   AI_RAW_8701.___________0040_1 := false;
   AI_RAW_8701.___________0040_2 := false;
   AI_RAW_8701.VALUE_COEF := 0.00617;
   AI_RAW_8801.revInfo.REV_BLOCK := 'UT00801';
   AI_RAW_8801.revInfo.REV_NUMBER := '001.000';
   AI_RAW_8801.revInfo.REV_DATE := '2024-04-09';
   AI_RAW_8801.revInfo.REV_AUTHOR := 'M. Gledhill';
   AI_RAW_8801.___________0010_0 := false;
   AI_RAW_8801.___________0010_1 := false;
   AI_RAW_8801.AI_CODE := 16#8801;
   AI_RAW_8801.___________0020_0 := false;
   AI_RAW_8801.___________0020_1 := false;
   AI_RAW_8801.RAW_MIN := -6000;
   AI_RAW_8801.RAW_MAX := 13000;
   AI_RAW_8801.RAW_DESC := 'Thermal Resistance - 3-wire (Ni100 climate - 618)';
   AI_RAW_8801.___________0030_1 := false;
   AI_RAW_8801.___________0030_2 := false;
   AI_RAW_8801.PARAM_TYPE := 16#08;
   AI_RAW_8801.PARAM_RANGE := 16#01;
   AI_RAW_8801.PARAM_COEF := 16#08;
   AI_RAW_8801.___________0040_1 := false;
   AI_RAW_8801.___________0040_2 := false;
   AI_RAW_8801.VALUE_COEF := 0.00618;
   AI_RAW_8901.revInfo.REV_BLOCK := 'UT00801';
   AI_RAW_8901.revInfo.REV_NUMBER := '001.000';
   AI_RAW_8901.revInfo.REV_DATE := '2024-04-09';
   AI_RAW_8901.revInfo.REV_AUTHOR := 'M. Gledhill';
   AI_RAW_8901.___________0010_0 := false;
   AI_RAW_8901.___________0010_1 := false;
   AI_RAW_8901.AI_CODE := 16#8901;
   AI_RAW_8901.___________0020_0 := false;
   AI_RAW_8901.___________0020_1 := false;
   AI_RAW_8901.RAW_MIN := -6000;
   AI_RAW_8901.RAW_MAX := 13000;
   AI_RAW_8901.RAW_DESC := 'Thermal Resistance - 3-wire (Ni100 climate - 672)';
   AI_RAW_8901.___________0030_1 := false;
   AI_RAW_8901.___________0030_2 := false;
   AI_RAW_8901.PARAM_TYPE := 16#08;
   AI_RAW_8901.PARAM_RANGE := 16#01;
   AI_RAW_8901.PARAM_COEF := 16#09;
   AI_RAW_8901.___________0040_1 := false;
   AI_RAW_8901.___________0040_2 := false;
   AI_RAW_8901.VALUE_COEF := 0.00672;
   AI_RAW_8703.revInfo.REV_BLOCK := 'UT00801';
   AI_RAW_8703.revInfo.REV_NUMBER := '001.000';
   AI_RAW_8703.revInfo.REV_DATE := '2024-04-09';
   AI_RAW_8703.revInfo.REV_AUTHOR := 'M. Gledhill';
   AI_RAW_8703.___________0010_0 := false;
   AI_RAW_8703.___________0010_1 := false;
   AI_RAW_8703.AI_CODE := 16#8703;
   AI_RAW_8703.___________0020_0 := false;
   AI_RAW_8703.___________0020_1 := false;
   AI_RAW_8703.RAW_MIN := -600;
   AI_RAW_8703.RAW_MAX := 1800;
   AI_RAW_8703.RAW_DESC := 'Thermal Resistance - 3-wire (Ni100 standard - 617)';
   AI_RAW_8703.___________0030_1 := false;
   AI_RAW_8703.___________0030_2 := false;
   AI_RAW_8703.PARAM_TYPE := 16#08;
   AI_RAW_8703.PARAM_RANGE := 16#03;
   AI_RAW_8703.PARAM_COEF := 16#07;
   AI_RAW_8703.___________0040_1 := false;
   AI_RAW_8703.___________0040_2 := false;
   AI_RAW_8703.VALUE_COEF := 0.00617;
   AI_RAW_8803.revInfo.REV_BLOCK := 'UT00801';
   AI_RAW_8803.revInfo.REV_NUMBER := '001.000';
   AI_RAW_8803.revInfo.REV_DATE := '2024-04-09';
   AI_RAW_8803.revInfo.REV_AUTHOR := 'M. Gledhill';
   AI_RAW_8803.___________0010_0 := false;
   AI_RAW_8803.___________0010_1 := false;
   AI_RAW_8803.AI_CODE := 16#8803;
   AI_RAW_8803.___________0020_0 := false;
   AI_RAW_8803.___________0020_1 := false;
   AI_RAW_8803.RAW_MIN := -600;
   AI_RAW_8803.RAW_MAX := 2500;
   AI_RAW_8803.RAW_DESC := 'Thermal Resistance - 3-wire (Ni100 standard - 618)';
   AI_RAW_8803.___________0030_1 := false;
   AI_RAW_8803.___________0030_2 := false;
   AI_RAW_8803.PARAM_TYPE := 16#08;
   AI_RAW_8803.PARAM_RANGE := 16#03;
   AI_RAW_8803.PARAM_COEF := 16#08;
   AI_RAW_8803.___________0040_1 := false;
   AI_RAW_8803.___________0040_2 := false;
   AI_RAW_8803.VALUE_COEF := 0.00618;
   AI_RAW_8903.revInfo.REV_BLOCK := 'UT00801';
   AI_RAW_8903.revInfo.REV_NUMBER := '001.000';
   AI_RAW_8903.revInfo.REV_DATE := '2024-04-09';
   AI_RAW_8903.revInfo.REV_AUTHOR := 'M. Gledhill';
   AI_RAW_8903.___________0010_0 := false;
   AI_RAW_8903.___________0010_1 := false;
   AI_RAW_8903.AI_CODE := 16#8903;
   AI_RAW_8903.___________0020_0 := false;
   AI_RAW_8903.___________0020_1 := false;
   AI_RAW_8903.RAW_MIN := -600;
   AI_RAW_8903.RAW_MAX := 2500;
   AI_RAW_8903.RAW_DESC := 'Thermal Resistance - 3-wire (Ni100 standard - 672)';
   AI_RAW_8903.___________0030_1 := false;
   AI_RAW_8903.___________0030_2 := false;
   AI_RAW_8903.PARAM_TYPE := 16#08;
   AI_RAW_8903.PARAM_RANGE := 16#03;
   AI_RAW_8903.PARAM_COEF := 16#09;
   AI_RAW_8903.___________0040_1 := false;
   AI_RAW_8903.___________0040_2 := false;
   AI_RAW_8903.VALUE_COEF := 0.00672;
   AI_RAW_8711.revInfo.REV_BLOCK := 'UT00801';
   AI_RAW_8711.revInfo.REV_NUMBER := '001.000';
   AI_RAW_8711.revInfo.REV_DATE := '2024-04-09';
   AI_RAW_8711.revInfo.REV_AUTHOR := 'M. Gledhill';
   AI_RAW_8711.___________0010_0 := false;
   AI_RAW_8711.___________0010_1 := false;
   AI_RAW_8711.AI_CODE := 16#8711;
   AI_RAW_8711.___________0020_0 := false;
   AI_RAW_8711.___________0020_1 := false;
   AI_RAW_8711.RAW_MIN := -6000;
   AI_RAW_8711.RAW_MAX := 13000;
   AI_RAW_8711.RAW_DESC := 'Thermal Resistance - 3-wire (Ni200 climate - 617)';
   AI_RAW_8711.___________0030_1 := false;
   AI_RAW_8711.___________0030_2 := false;
   AI_RAW_8711.PARAM_TYPE := 16#08;
   AI_RAW_8711.PARAM_RANGE := 16#11;
   AI_RAW_8711.PARAM_COEF := 16#07;
   AI_RAW_8711.___________0040_1 := false;
   AI_RAW_8711.___________0040_2 := false;
   AI_RAW_8711.VALUE_COEF := 0.00617;
   AI_RAW_8811.revInfo.REV_BLOCK := 'UT00801';
   AI_RAW_8811.revInfo.REV_NUMBER := '001.000';
   AI_RAW_8811.revInfo.REV_DATE := '2024-04-09';
   AI_RAW_8811.revInfo.REV_AUTHOR := 'M. Gledhill';
   AI_RAW_8811.___________0010_0 := false;
   AI_RAW_8811.___________0010_1 := false;
   AI_RAW_8811.AI_CODE := 16#8811;
   AI_RAW_8811.___________0020_0 := false;
   AI_RAW_8811.___________0020_1 := false;
   AI_RAW_8811.RAW_MIN := -6000;
   AI_RAW_8811.RAW_MAX := 13000;
   AI_RAW_8811.RAW_DESC := 'Thermal Resistance - 3-wire (Ni200 climate - 618)';
   AI_RAW_8811.___________0030_1 := false;
   AI_RAW_8811.___________0030_2 := false;
   AI_RAW_8811.PARAM_TYPE := 16#08;
   AI_RAW_8811.PARAM_RANGE := 16#11;
   AI_RAW_8811.PARAM_COEF := 16#08;
   AI_RAW_8811.___________0040_1 := false;
   AI_RAW_8811.___________0040_2 := false;
   AI_RAW_8811.VALUE_COEF := 0.00618;
   AI_RAW_8911.revInfo.REV_BLOCK := 'UT00801';
   AI_RAW_8911.revInfo.REV_NUMBER := '001.000';
   AI_RAW_8911.revInfo.REV_DATE := '2024-04-09';
   AI_RAW_8911.revInfo.REV_AUTHOR := 'M. Gledhill';
   AI_RAW_8911.___________0010_0 := false;
   AI_RAW_8911.___________0010_1 := false;
   AI_RAW_8911.AI_CODE := 16#8911;
   AI_RAW_8911.___________0020_0 := false;
   AI_RAW_8911.___________0020_1 := false;
   AI_RAW_8911.RAW_MIN := -6000;
   AI_RAW_8911.RAW_MAX := 13000;
   AI_RAW_8911.RAW_DESC := 'Thermal Resistance - 3-wire (Ni200 climate - 672)';
   AI_RAW_8911.___________0030_1 := false;
   AI_RAW_8911.___________0030_2 := false;
   AI_RAW_8911.PARAM_TYPE := 16#08;
   AI_RAW_8911.PARAM_RANGE := 16#11;
   AI_RAW_8911.PARAM_COEF := 16#09;
   AI_RAW_8911.___________0040_1 := false;
   AI_RAW_8911.___________0040_2 := false;
   AI_RAW_8911.VALUE_COEF := 0.00672;
   AI_RAW_8710.revInfo.REV_BLOCK := 'UT00801';
   AI_RAW_8710.revInfo.REV_NUMBER := '001.000';
   AI_RAW_8710.revInfo.REV_DATE := '2024-04-09';
   AI_RAW_8710.revInfo.REV_AUTHOR := 'M. Gledhill';
   AI_RAW_8710.___________0010_0 := false;
   AI_RAW_8710.___________0010_1 := false;
   AI_RAW_8710.AI_CODE := 16#8710;
   AI_RAW_8710.___________0020_0 := false;
   AI_RAW_8710.___________0020_1 := false;
   AI_RAW_8710.RAW_MIN := -600;
   AI_RAW_8710.RAW_MAX := 1800;
   AI_RAW_8710.RAW_DESC := 'Thermal Resistance - 3-wire (Ni200 standard - 617)';
   AI_RAW_8710.___________0030_1 := false;
   AI_RAW_8710.___________0030_2 := false;
   AI_RAW_8710.PARAM_TYPE := 16#08;
   AI_RAW_8710.PARAM_RANGE := 16#10;
   AI_RAW_8710.PARAM_COEF := 16#07;
   AI_RAW_8710.___________0040_1 := false;
   AI_RAW_8710.___________0040_2 := false;
   AI_RAW_8710.VALUE_COEF := 0.00617;
   AI_RAW_8810.revInfo.REV_BLOCK := 'UT00801';
   AI_RAW_8810.revInfo.REV_NUMBER := '001.000';
   AI_RAW_8810.revInfo.REV_DATE := '2024-04-09';
   AI_RAW_8810.revInfo.REV_AUTHOR := 'M. Gledhill';
   AI_RAW_8810.___________0010_0 := false;
   AI_RAW_8810.___________0010_1 := false;
   AI_RAW_8810.AI_CODE := 16#8810;
   AI_RAW_8810.___________0020_0 := false;
   AI_RAW_8810.___________0020_1 := false;
   AI_RAW_8810.RAW_MIN := -600;
   AI_RAW_8810.RAW_MAX := 2500;
   AI_RAW_8810.RAW_DESC := 'Thermal Resistance - 3-wire (Ni200 standard - 618)';
   AI_RAW_8810.___________0030_1 := false;
   AI_RAW_8810.___________0030_2 := false;
   AI_RAW_8810.PARAM_TYPE := 16#08;
   AI_RAW_8810.PARAM_RANGE := 16#10;
   AI_RAW_8810.PARAM_COEF := 16#08;
   AI_RAW_8810.___________0040_1 := false;
   AI_RAW_8810.___________0040_2 := false;
   AI_RAW_8810.VALUE_COEF := 0.00618;
   AI_RAW_8910.revInfo.REV_BLOCK := 'UT00801';
   AI_RAW_8910.revInfo.REV_NUMBER := '001.000';
   AI_RAW_8910.revInfo.REV_DATE := '2024-04-09';
   AI_RAW_8910.revInfo.REV_AUTHOR := 'M. Gledhill';
   AI_RAW_8910.___________0010_0 := false;
   AI_RAW_8910.___________0010_1 := false;
   AI_RAW_8910.AI_CODE := 16#8910;
   AI_RAW_8910.___________0020_0 := false;
   AI_RAW_8910.___________0020_1 := false;
   AI_RAW_8910.RAW_MIN := -600;
   AI_RAW_8910.RAW_MAX := 2500;
   AI_RAW_8910.RAW_DESC := 'Thermal Resistance - 3-wire (Ni200 standard - 672)';
   AI_RAW_8910.___________0030_1 := false;
   AI_RAW_8910.___________0030_2 := false;
   AI_RAW_8910.PARAM_TYPE := 16#08;
   AI_RAW_8910.PARAM_RANGE := 16#10;
   AI_RAW_8910.PARAM_COEF := 16#09;
   AI_RAW_8910.___________0040_1 := false;
   AI_RAW_8910.___________0040_2 := false;
   AI_RAW_8910.VALUE_COEF := 0.00672;
   AI_RAW_8713.revInfo.REV_BLOCK := 'UT00801';
   AI_RAW_8713.revInfo.REV_NUMBER := '001.000';
   AI_RAW_8713.revInfo.REV_DATE := '2024-04-09';
   AI_RAW_8713.revInfo.REV_AUTHOR := 'M. Gledhill';
   AI_RAW_8713.___________0010_0 := false;
   AI_RAW_8713.___________0010_1 := false;
   AI_RAW_8713.AI_CODE := 16#8713;
   AI_RAW_8713.___________0020_0 := false;
   AI_RAW_8713.___________0020_1 := false;
   AI_RAW_8713.RAW_MIN := -6000;
   AI_RAW_8713.RAW_MAX := 13000;
   AI_RAW_8713.RAW_DESC := 'Thermal Resistance - 3-wire (Ni500 climate - 617)';
   AI_RAW_8713.___________0030_1 := false;
   AI_RAW_8713.___________0030_2 := false;
   AI_RAW_8713.PARAM_TYPE := 16#08;
   AI_RAW_8713.PARAM_RANGE := 16#13;
   AI_RAW_8713.PARAM_COEF := 16#07;
   AI_RAW_8713.___________0040_1 := false;
   AI_RAW_8713.___________0040_2 := false;
   AI_RAW_8713.VALUE_COEF := 0.00617;
   AI_RAW_8813.revInfo.REV_BLOCK := 'UT00801';
   AI_RAW_8813.revInfo.REV_NUMBER := '001.000';
   AI_RAW_8813.revInfo.REV_DATE := '2024-04-09';
   AI_RAW_8813.revInfo.REV_AUTHOR := 'M. Gledhill';
   AI_RAW_8813.___________0010_0 := false;
   AI_RAW_8813.___________0010_1 := false;
   AI_RAW_8813.AI_CODE := 16#8813;
   AI_RAW_8813.___________0020_0 := false;
   AI_RAW_8813.___________0020_1 := false;
   AI_RAW_8813.RAW_MIN := -6000;
   AI_RAW_8813.RAW_MAX := 13000;
   AI_RAW_8813.RAW_DESC := 'Thermal Resistance - 3-wire (Ni500 climate - 618)';
   AI_RAW_8813.___________0030_1 := false;
   AI_RAW_8813.___________0030_2 := false;
   AI_RAW_8813.PARAM_TYPE := 16#08;
   AI_RAW_8813.PARAM_RANGE := 16#13;
   AI_RAW_8813.PARAM_COEF := 16#08;
   AI_RAW_8813.___________0040_1 := false;
   AI_RAW_8813.___________0040_2 := false;
   AI_RAW_8813.VALUE_COEF := 0.00618;
   AI_RAW_8913.revInfo.REV_BLOCK := 'UT00801';
   AI_RAW_8913.revInfo.REV_NUMBER := '001.000';
   AI_RAW_8913.revInfo.REV_DATE := '2024-04-09';
   AI_RAW_8913.revInfo.REV_AUTHOR := 'M. Gledhill';
   AI_RAW_8913.___________0010_0 := false;
   AI_RAW_8913.___________0010_1 := false;
   AI_RAW_8913.AI_CODE := 16#8913;
   AI_RAW_8913.___________0020_0 := false;
   AI_RAW_8913.___________0020_1 := false;
   AI_RAW_8913.RAW_MIN := -6000;
   AI_RAW_8913.RAW_MAX := 13000;
   AI_RAW_8913.RAW_DESC := 'Thermal Resistance - 3-wire (Ni500 climate - 672)';
   AI_RAW_8913.___________0030_1 := false;
   AI_RAW_8913.___________0030_2 := false;
   AI_RAW_8913.PARAM_TYPE := 16#08;
   AI_RAW_8913.PARAM_RANGE := 16#13;
   AI_RAW_8913.PARAM_COEF := 16#09;
   AI_RAW_8913.___________0040_1 := false;
   AI_RAW_8913.___________0040_2 := false;
   AI_RAW_8913.VALUE_COEF := 0.00672;
   AI_RAW_8712.revInfo.REV_BLOCK := 'UT00801';
   AI_RAW_8712.revInfo.REV_NUMBER := '001.000';
   AI_RAW_8712.revInfo.REV_DATE := '2024-04-09';
   AI_RAW_8712.revInfo.REV_AUTHOR := 'M. Gledhill';
   AI_RAW_8712.___________0010_0 := false;
   AI_RAW_8712.___________0010_1 := false;
   AI_RAW_8712.AI_CODE := 16#8712;
   AI_RAW_8712.___________0020_0 := false;
   AI_RAW_8712.___________0020_1 := false;
   AI_RAW_8712.RAW_MIN := -600;
   AI_RAW_8712.RAW_MAX := 1800;
   AI_RAW_8712.RAW_DESC := 'Thermal Resistance - 3-wire (Ni500 standard - 617)';
   AI_RAW_8712.___________0030_1 := false;
   AI_RAW_8712.___________0030_2 := false;
   AI_RAW_8712.PARAM_TYPE := 16#08;
   AI_RAW_8712.PARAM_RANGE := 16#12;
   AI_RAW_8712.PARAM_COEF := 16#07;
   AI_RAW_8712.___________0040_1 := false;
   AI_RAW_8712.___________0040_2 := false;
   AI_RAW_8712.VALUE_COEF := 0.00617;
   AI_RAW_8812.revInfo.REV_BLOCK := 'UT00801';
   AI_RAW_8812.revInfo.REV_NUMBER := '001.000';
   AI_RAW_8812.revInfo.REV_DATE := '2024-04-09';
   AI_RAW_8812.revInfo.REV_AUTHOR := 'M. Gledhill';
   AI_RAW_8812.___________0010_0 := false;
   AI_RAW_8812.___________0010_1 := false;
   AI_RAW_8812.AI_CODE := 16#8812;
   AI_RAW_8812.___________0020_0 := false;
   AI_RAW_8812.___________0020_1 := false;
   AI_RAW_8812.RAW_MIN := -600;
   AI_RAW_8812.RAW_MAX := 2500;
   AI_RAW_8812.RAW_DESC := 'Thermal Resistance - 3-wire (Ni500 standard - 618)';
   AI_RAW_8812.___________0030_1 := false;
   AI_RAW_8812.___________0030_2 := false;
   AI_RAW_8812.PARAM_TYPE := 16#08;
   AI_RAW_8812.PARAM_RANGE := 16#12;
   AI_RAW_8812.PARAM_COEF := 16#08;
   AI_RAW_8812.___________0040_1 := false;
   AI_RAW_8812.___________0040_2 := false;
   AI_RAW_8812.VALUE_COEF := 0.00618;
   AI_RAW_8912.revInfo.REV_BLOCK := 'UT00801';
   AI_RAW_8912.revInfo.REV_NUMBER := '001.000';
   AI_RAW_8912.revInfo.REV_DATE := '2024-04-09';
   AI_RAW_8912.revInfo.REV_AUTHOR := 'M. Gledhill';
   AI_RAW_8912.___________0010_0 := false;
   AI_RAW_8912.___________0010_1 := false;
   AI_RAW_8912.AI_CODE := 16#8912;
   AI_RAW_8912.___________0020_0 := false;
   AI_RAW_8912.___________0020_1 := false;
   AI_RAW_8912.RAW_MIN := -600;
   AI_RAW_8912.RAW_MAX := 2500;
   AI_RAW_8912.RAW_DESC := 'Thermal Resistance - 3-wire (Ni500 standard - 672)';
   AI_RAW_8912.___________0030_1 := false;
   AI_RAW_8912.___________0030_2 := false;
   AI_RAW_8912.PARAM_TYPE := 16#08;
   AI_RAW_8912.PARAM_RANGE := 16#12;
   AI_RAW_8912.PARAM_COEF := 16#09;
   AI_RAW_8912.___________0040_1 := false;
   AI_RAW_8912.___________0040_2 := false;
   AI_RAW_8912.VALUE_COEF := 0.00672;
   AI_RAW_870A.revInfo.REV_BLOCK := 'UT00801';
   AI_RAW_870A.revInfo.REV_NUMBER := '001.000';
   AI_RAW_870A.revInfo.REV_DATE := '2024-04-09';
   AI_RAW_870A.revInfo.REV_AUTHOR := 'M. Gledhill';
   AI_RAW_870A.___________0010_0 := false;
   AI_RAW_870A.___________0010_1 := false;
   AI_RAW_870A.AI_CODE := 16#870A;
   AI_RAW_870A.___________0020_0 := false;
   AI_RAW_870A.___________0020_1 := false;
   AI_RAW_870A.RAW_MIN := -6000;
   AI_RAW_870A.RAW_MAX := 13000;
   AI_RAW_870A.RAW_DESC := 'Thermal Resistance - 3-wire (Ni1000 climate - 617)';
   AI_RAW_870A.___________0030_1 := false;
   AI_RAW_870A.___________0030_2 := false;
   AI_RAW_870A.PARAM_TYPE := 16#08;
   AI_RAW_870A.PARAM_RANGE := 16#0A;
   AI_RAW_870A.PARAM_COEF := 16#07;
   AI_RAW_870A.___________0040_1 := false;
   AI_RAW_870A.___________0040_2 := false;
   AI_RAW_870A.VALUE_COEF := 0.00617;
   AI_RAW_880A.revInfo.REV_BLOCK := 'UT00801';
   AI_RAW_880A.revInfo.REV_NUMBER := '001.000';
   AI_RAW_880A.revInfo.REV_DATE := '2024-04-09';
   AI_RAW_880A.revInfo.REV_AUTHOR := 'M. Gledhill';
   AI_RAW_880A.___________0010_0 := false;
   AI_RAW_880A.___________0010_1 := false;
   AI_RAW_880A.AI_CODE := 16#880A;
   AI_RAW_880A.___________0020_0 := false;
   AI_RAW_880A.___________0020_1 := false;
   AI_RAW_880A.RAW_MIN := -6000;
   AI_RAW_880A.RAW_MAX := 13000;
   AI_RAW_880A.RAW_DESC := 'Thermal Resistance - 3-wire (Ni1000 climate - 618)';
   AI_RAW_880A.___________0030_1 := false;
   AI_RAW_880A.___________0030_2 := false;
   AI_RAW_880A.PARAM_TYPE := 16#08;
   AI_RAW_880A.PARAM_RANGE := 16#0A;
   AI_RAW_880A.PARAM_COEF := 16#08;
   AI_RAW_880A.___________0040_1 := false;
   AI_RAW_880A.___________0040_2 := false;
   AI_RAW_880A.VALUE_COEF := 0.00618;
   AI_RAW_890A.revInfo.REV_BLOCK := 'UT00801';
   AI_RAW_890A.revInfo.REV_NUMBER := '001.000';
   AI_RAW_890A.revInfo.REV_DATE := '2024-04-09';
   AI_RAW_890A.revInfo.REV_AUTHOR := 'M. Gledhill';
   AI_RAW_890A.___________0010_0 := false;
   AI_RAW_890A.___________0010_1 := false;
   AI_RAW_890A.AI_CODE := 16#890A;
   AI_RAW_890A.___________0020_0 := false;
   AI_RAW_890A.___________0020_1 := false;
   AI_RAW_890A.RAW_MIN := -6000;
   AI_RAW_890A.RAW_MAX := 13000;
   AI_RAW_890A.RAW_DESC := 'Thermal Resistance - 3-wire (Ni1000 climate - 672)';
   AI_RAW_890A.___________0030_1 := false;
   AI_RAW_890A.___________0030_2 := false;
   AI_RAW_890A.PARAM_TYPE := 16#08;
   AI_RAW_890A.PARAM_RANGE := 16#0A;
   AI_RAW_890A.PARAM_COEF := 16#09;
   AI_RAW_890A.___________0040_1 := false;
   AI_RAW_890A.___________0040_2 := false;
   AI_RAW_890A.VALUE_COEF := 0.00672;
   AI_RAW_8706.revInfo.REV_BLOCK := 'UT00801';
   AI_RAW_8706.revInfo.REV_NUMBER := '001.000';
   AI_RAW_8706.revInfo.REV_DATE := '2024-04-09';
   AI_RAW_8706.revInfo.REV_AUTHOR := 'M. Gledhill';
   AI_RAW_8706.___________0010_0 := false;
   AI_RAW_8706.___________0010_1 := false;
   AI_RAW_8706.AI_CODE := 16#8706;
   AI_RAW_8706.___________0020_0 := false;
   AI_RAW_8706.___________0020_1 := false;
   AI_RAW_8706.RAW_MIN := -600;
   AI_RAW_8706.RAW_MAX := 1800;
   AI_RAW_8706.RAW_DESC := 'Thermal Resistance - 3-wire (Ni1000 standard - 617)';
   AI_RAW_8706.___________0030_1 := false;
   AI_RAW_8706.___________0030_2 := false;
   AI_RAW_8706.PARAM_TYPE := 16#08;
   AI_RAW_8706.PARAM_RANGE := 16#06;
   AI_RAW_8706.PARAM_COEF := 16#07;
   AI_RAW_8706.___________0040_1 := false;
   AI_RAW_8706.___________0040_2 := false;
   AI_RAW_8706.VALUE_COEF := 0.00617;
   AI_RAW_8806.revInfo.REV_BLOCK := 'UT00801';
   AI_RAW_8806.revInfo.REV_NUMBER := '001.000';
   AI_RAW_8806.revInfo.REV_DATE := '2024-04-09';
   AI_RAW_8806.revInfo.REV_AUTHOR := 'M. Gledhill';
   AI_RAW_8806.___________0010_0 := false;
   AI_RAW_8806.___________0010_1 := false;
   AI_RAW_8806.AI_CODE := 16#8806;
   AI_RAW_8806.___________0020_0 := false;
   AI_RAW_8806.___________0020_1 := false;
   AI_RAW_8806.RAW_MIN := -600;
   AI_RAW_8806.RAW_MAX := 2500;
   AI_RAW_8806.RAW_DESC := 'Thermal Resistance - 3-wire (Ni1000 standard - 618)';
   AI_RAW_8806.___________0030_1 := false;
   AI_RAW_8806.___________0030_2 := false;
   AI_RAW_8806.PARAM_TYPE := 16#08;
   AI_RAW_8806.PARAM_RANGE := 16#06;
   AI_RAW_8806.PARAM_COEF := 16#08;
   AI_RAW_8806.___________0040_1 := false;
   AI_RAW_8806.___________0040_2 := false;
   AI_RAW_8806.VALUE_COEF := 0.00618;
   AI_RAW_8906.revInfo.REV_BLOCK := 'UT00801';
   AI_RAW_8906.revInfo.REV_NUMBER := '001.000';
   AI_RAW_8906.revInfo.REV_DATE := '2024-04-09';
   AI_RAW_8906.revInfo.REV_AUTHOR := 'M. Gledhill';
   AI_RAW_8906.___________0010_0 := false;
   AI_RAW_8906.___________0010_1 := false;
   AI_RAW_8906.AI_CODE := 16#8906;
   AI_RAW_8906.___________0020_0 := false;
   AI_RAW_8906.___________0020_1 := false;
   AI_RAW_8906.RAW_MIN := -600;
   AI_RAW_8906.RAW_MAX := 2500;
   AI_RAW_8906.RAW_DESC := 'Thermal Resistance - 3-wire (Ni1000 standard - 672)';
   AI_RAW_8906.___________0030_1 := false;
   AI_RAW_8906.___________0030_2 := false;
   AI_RAW_8906.PARAM_TYPE := 16#08;
   AI_RAW_8906.PARAM_RANGE := 16#06;
   AI_RAW_8906.PARAM_COEF := 16#09;
   AI_RAW_8906.___________0040_1 := false;
   AI_RAW_8906.___________0040_2 := false;
   AI_RAW_8906.VALUE_COEF := 0.00672;
   AI_RAW_8015.revInfo.REV_BLOCK := 'UT00801';
   AI_RAW_8015.revInfo.REV_NUMBER := '001.000';
   AI_RAW_8015.revInfo.REV_DATE := '2024-04-09';
   AI_RAW_8015.revInfo.REV_AUTHOR := 'M. Gledhill';
   AI_RAW_8015.___________0010_0 := false;
   AI_RAW_8015.___________0010_1 := false;
   AI_RAW_8015.AI_CODE := 16#8015;
   AI_RAW_8015.___________0020_0 := false;
   AI_RAW_8015.___________0020_1 := false;
   AI_RAW_8015.RAW_MIN := -12000;
   AI_RAW_8015.RAW_MAX := 13000;
   AI_RAW_8015.RAW_DESC := 'Thermal Resistance - 3-wire (Pt10 climate - 3851)';
   AI_RAW_8015.___________0030_1 := false;
   AI_RAW_8015.___________0030_2 := false;
   AI_RAW_8015.PARAM_TYPE := 16#08;
   AI_RAW_8015.PARAM_RANGE := 16#15;
   AI_RAW_8015.PARAM_COEF := 16#00;
   AI_RAW_8015.___________0040_1 := false;
   AI_RAW_8015.___________0040_2 := false;
   AI_RAW_8015.VALUE_COEF := 0.003851;
   AI_RAW_8215.revInfo.REV_BLOCK := 'UT00801';
   AI_RAW_8215.revInfo.REV_NUMBER := '001.000';
   AI_RAW_8215.revInfo.REV_DATE := '2024-04-09';
   AI_RAW_8215.revInfo.REV_AUTHOR := 'M. Gledhill';
   AI_RAW_8215.___________0010_0 := false;
   AI_RAW_8215.___________0010_1 := false;
   AI_RAW_8215.AI_CODE := 16#8215;
   AI_RAW_8215.___________0020_0 := false;
   AI_RAW_8215.___________0020_1 := false;
   AI_RAW_8215.RAW_MIN := -12000;
   AI_RAW_8215.RAW_MAX := 13000;
   AI_RAW_8215.RAW_DESC := 'Thermal Resistance - 3-wire (Pt10 climate - 3902)';
   AI_RAW_8215.___________0030_1 := false;
   AI_RAW_8215.___________0030_2 := false;
   AI_RAW_8215.PARAM_TYPE := 16#08;
   AI_RAW_8215.PARAM_RANGE := 16#15;
   AI_RAW_8215.PARAM_COEF := 16#02;
   AI_RAW_8215.___________0040_1 := false;
   AI_RAW_8215.___________0040_2 := false;
   AI_RAW_8215.VALUE_COEF := 0.003902;
   AI_RAW_8515.revInfo.REV_BLOCK := 'UT00801';
   AI_RAW_8515.revInfo.REV_NUMBER := '001.000';
   AI_RAW_8515.revInfo.REV_DATE := '2024-04-09';
   AI_RAW_8515.revInfo.REV_AUTHOR := 'M. Gledhill';
   AI_RAW_8515.___________0010_0 := false;
   AI_RAW_8515.___________0010_1 := false;
   AI_RAW_8515.AI_CODE := 16#8515;
   AI_RAW_8515.___________0020_0 := false;
   AI_RAW_8515.___________0020_1 := false;
   AI_RAW_8515.RAW_MIN := -12000;
   AI_RAW_8515.RAW_MAX := 13000;
   AI_RAW_8515.RAW_DESC := 'Thermal Resistance - 3-wire (Pt10 climate - 391)';
   AI_RAW_8515.___________0030_1 := false;
   AI_RAW_8515.___________0030_2 := false;
   AI_RAW_8515.PARAM_TYPE := 16#08;
   AI_RAW_8515.PARAM_RANGE := 16#15;
   AI_RAW_8515.PARAM_COEF := 16#05;
   AI_RAW_8515.___________0040_1 := false;
   AI_RAW_8515.___________0040_2 := false;
   AI_RAW_8515.VALUE_COEF := 0.00391;
   AI_RAW_8115.revInfo.REV_BLOCK := 'UT00801';
   AI_RAW_8115.revInfo.REV_NUMBER := '001.000';
   AI_RAW_8115.revInfo.REV_DATE := '2024-04-09';
   AI_RAW_8115.revInfo.REV_AUTHOR := 'M. Gledhill';
   AI_RAW_8115.___________0010_0 := false;
   AI_RAW_8115.___________0010_1 := false;
   AI_RAW_8115.AI_CODE := 16#8115;
   AI_RAW_8115.___________0020_0 := false;
   AI_RAW_8115.___________0020_1 := false;
   AI_RAW_8115.RAW_MIN := -12000;
   AI_RAW_8115.RAW_MAX := 13000;
   AI_RAW_8115.RAW_DESC := 'Thermal Resistance - 3-wire (Pt10 climate - 3916)';
   AI_RAW_8115.___________0030_1 := false;
   AI_RAW_8115.___________0030_2 := false;
   AI_RAW_8115.PARAM_TYPE := 16#08;
   AI_RAW_8115.PARAM_RANGE := 16#15;
   AI_RAW_8115.PARAM_COEF := 16#01;
   AI_RAW_8115.___________0040_1 := false;
   AI_RAW_8115.___________0040_2 := false;
   AI_RAW_8115.VALUE_COEF := 0.003916;
   AI_RAW_8315.revInfo.REV_BLOCK := 'UT00801';
   AI_RAW_8315.revInfo.REV_NUMBER := '001.000';
   AI_RAW_8315.revInfo.REV_DATE := '2024-04-09';
   AI_RAW_8315.revInfo.REV_AUTHOR := 'M. Gledhill';
   AI_RAW_8315.___________0010_0 := false;
   AI_RAW_8315.___________0010_1 := false;
   AI_RAW_8315.AI_CODE := 16#8315;
   AI_RAW_8315.___________0020_0 := false;
   AI_RAW_8315.___________0020_1 := false;
   AI_RAW_8315.RAW_MIN := -12000;
   AI_RAW_8315.RAW_MAX := 13000;
   AI_RAW_8315.RAW_DESC := 'Thermal Resistance - 3-wire (Pt10 climate - 392)';
   AI_RAW_8315.___________0030_1 := false;
   AI_RAW_8315.___________0030_2 := false;
   AI_RAW_8315.PARAM_TYPE := 16#08;
   AI_RAW_8315.PARAM_RANGE := 16#15;
   AI_RAW_8315.PARAM_COEF := 16#03;
   AI_RAW_8315.___________0040_1 := false;
   AI_RAW_8315.___________0040_2 := false;
   AI_RAW_8315.VALUE_COEF := 0.00392;
   AI_RAW_8014.revInfo.REV_BLOCK := 'UT00801';
   AI_RAW_8014.revInfo.REV_NUMBER := '001.000';
   AI_RAW_8014.revInfo.REV_DATE := '2024-04-09';
   AI_RAW_8014.revInfo.REV_AUTHOR := 'M. Gledhill';
   AI_RAW_8014.___________0010_0 := false;
   AI_RAW_8014.___________0010_1 := false;
   AI_RAW_8014.AI_CODE := 16#8014;
   AI_RAW_8014.___________0020_0 := false;
   AI_RAW_8014.___________0020_1 := false;
   AI_RAW_8014.RAW_MIN := -2000;
   AI_RAW_8014.RAW_MAX := 8500;
   AI_RAW_8014.RAW_DESC := 'Thermal Resistance - 3-wire (Pt10 standard - 3851)';
   AI_RAW_8014.___________0030_1 := false;
   AI_RAW_8014.___________0030_2 := false;
   AI_RAW_8014.PARAM_TYPE := 16#08;
   AI_RAW_8014.PARAM_RANGE := 16#14;
   AI_RAW_8014.PARAM_COEF := 16#00;
   AI_RAW_8014.___________0040_1 := false;
   AI_RAW_8014.___________0040_2 := false;
   AI_RAW_8014.VALUE_COEF := 0.003851;
   AI_RAW_8214.revInfo.REV_BLOCK := 'UT00801';
   AI_RAW_8214.revInfo.REV_NUMBER := '001.000';
   AI_RAW_8214.revInfo.REV_DATE := '2024-04-09';
   AI_RAW_8214.revInfo.REV_AUTHOR := 'M. Gledhill';
   AI_RAW_8214.___________0010_0 := false;
   AI_RAW_8214.___________0010_1 := false;
   AI_RAW_8214.AI_CODE := 16#8214;
   AI_RAW_8214.___________0020_0 := false;
   AI_RAW_8214.___________0020_1 := false;
   AI_RAW_8214.RAW_MIN := -2000;
   AI_RAW_8214.RAW_MAX := 8500;
   AI_RAW_8214.RAW_DESC := 'Thermal Resistance - 3-wire (Pt10 standard - 3902)';
   AI_RAW_8214.___________0030_1 := false;
   AI_RAW_8214.___________0030_2 := false;
   AI_RAW_8214.PARAM_TYPE := 16#08;
   AI_RAW_8214.PARAM_RANGE := 16#14;
   AI_RAW_8214.PARAM_COEF := 16#02;
   AI_RAW_8214.___________0040_1 := false;
   AI_RAW_8214.___________0040_2 := false;
   AI_RAW_8214.VALUE_COEF := 0.003902;
   AI_RAW_8514.revInfo.REV_BLOCK := 'UT00801';
   AI_RAW_8514.revInfo.REV_NUMBER := '001.000';
   AI_RAW_8514.revInfo.REV_DATE := '2024-04-09';
   AI_RAW_8514.revInfo.REV_AUTHOR := 'M. Gledhill';
   AI_RAW_8514.___________0010_0 := false;
   AI_RAW_8514.___________0010_1 := false;
   AI_RAW_8514.AI_CODE := 16#8514;
   AI_RAW_8514.___________0020_0 := false;
   AI_RAW_8514.___________0020_1 := false;
   AI_RAW_8514.RAW_MIN := -2000;
   AI_RAW_8514.RAW_MAX := 8500;
   AI_RAW_8514.RAW_DESC := 'Thermal Resistance - 3-wire (Pt10 standard - 391)';
   AI_RAW_8514.___________0030_1 := false;
   AI_RAW_8514.___________0030_2 := false;
   AI_RAW_8514.PARAM_TYPE := 16#08;
   AI_RAW_8514.PARAM_RANGE := 16#14;
   AI_RAW_8514.PARAM_COEF := 16#05;
   AI_RAW_8514.___________0040_1 := false;
   AI_RAW_8514.___________0040_2 := false;
   AI_RAW_8514.VALUE_COEF := 0.00391;
   AI_RAW_8114.revInfo.REV_BLOCK := 'UT00801';
   AI_RAW_8114.revInfo.REV_NUMBER := '001.000';
   AI_RAW_8114.revInfo.REV_DATE := '2024-04-09';
   AI_RAW_8114.revInfo.REV_AUTHOR := 'M. Gledhill';
   AI_RAW_8114.___________0010_0 := false;
   AI_RAW_8114.___________0010_1 := false;
   AI_RAW_8114.AI_CODE := 16#8114;
   AI_RAW_8114.___________0020_0 := false;
   AI_RAW_8114.___________0020_1 := false;
   AI_RAW_8114.RAW_MIN := -2000;
   AI_RAW_8114.RAW_MAX := 8500;
   AI_RAW_8114.RAW_DESC := 'Thermal Resistance - 3-wire (Pt10 standard - 3916)';
   AI_RAW_8114.___________0030_1 := false;
   AI_RAW_8114.___________0030_2 := false;
   AI_RAW_8114.PARAM_TYPE := 16#08;
   AI_RAW_8114.PARAM_RANGE := 16#14;
   AI_RAW_8114.PARAM_COEF := 16#01;
   AI_RAW_8114.___________0040_1 := false;
   AI_RAW_8114.___________0040_2 := false;
   AI_RAW_8114.VALUE_COEF := 0.003916;
   AI_RAW_8314.revInfo.REV_BLOCK := 'UT00801';
   AI_RAW_8314.revInfo.REV_NUMBER := '001.000';
   AI_RAW_8314.revInfo.REV_DATE := '2024-04-09';
   AI_RAW_8314.revInfo.REV_AUTHOR := 'M. Gledhill';
   AI_RAW_8314.___________0010_0 := false;
   AI_RAW_8314.___________0010_1 := false;
   AI_RAW_8314.AI_CODE := 16#8314;
   AI_RAW_8314.___________0020_0 := false;
   AI_RAW_8314.___________0020_1 := false;
   AI_RAW_8314.RAW_MIN := -2000;
   AI_RAW_8314.RAW_MAX := 8500;
   AI_RAW_8314.RAW_DESC := 'Thermal Resistance - 3-wire (Pt10 standard - 392)';
   AI_RAW_8314.___________0030_1 := false;
   AI_RAW_8314.___________0030_2 := false;
   AI_RAW_8314.PARAM_TYPE := 16#08;
   AI_RAW_8314.PARAM_RANGE := 16#14;
   AI_RAW_8314.PARAM_COEF := 16#03;
   AI_RAW_8314.___________0040_1 := false;
   AI_RAW_8314.___________0040_2 := false;
   AI_RAW_8314.VALUE_COEF := 0.00392;
   AI_RAW_8017.revInfo.REV_BLOCK := 'UT00801';
   AI_RAW_8017.revInfo.REV_NUMBER := '001.000';
   AI_RAW_8017.revInfo.REV_DATE := '2024-04-09';
   AI_RAW_8017.revInfo.REV_AUTHOR := 'M. Gledhill';
   AI_RAW_8017.___________0010_0 := false;
   AI_RAW_8017.___________0010_1 := false;
   AI_RAW_8017.AI_CODE := 16#8017;
   AI_RAW_8017.___________0020_0 := false;
   AI_RAW_8017.___________0020_1 := false;
   AI_RAW_8017.RAW_MIN := -12000;
   AI_RAW_8017.RAW_MAX := 13000;
   AI_RAW_8017.RAW_DESC := 'Thermal Resistance - 3-wire (Pt50 climate - 3851)';
   AI_RAW_8017.___________0030_1 := false;
   AI_RAW_8017.___________0030_2 := false;
   AI_RAW_8017.PARAM_TYPE := 16#08;
   AI_RAW_8017.PARAM_RANGE := 16#17;
   AI_RAW_8017.PARAM_COEF := 16#00;
   AI_RAW_8017.___________0040_1 := false;
   AI_RAW_8017.___________0040_2 := false;
   AI_RAW_8017.VALUE_COEF := 0.003851;
   AI_RAW_8217.revInfo.REV_BLOCK := 'UT00801';
   AI_RAW_8217.revInfo.REV_NUMBER := '001.000';
   AI_RAW_8217.revInfo.REV_DATE := '2024-04-09';
   AI_RAW_8217.revInfo.REV_AUTHOR := 'M. Gledhill';
   AI_RAW_8217.___________0010_0 := false;
   AI_RAW_8217.___________0010_1 := false;
   AI_RAW_8217.AI_CODE := 16#8217;
   AI_RAW_8217.___________0020_0 := false;
   AI_RAW_8217.___________0020_1 := false;
   AI_RAW_8217.RAW_MIN := -12000;
   AI_RAW_8217.RAW_MAX := 13000;
   AI_RAW_8217.RAW_DESC := 'Thermal Resistance - 3-wire (Pt50 climate - 3902)';
   AI_RAW_8217.___________0030_1 := false;
   AI_RAW_8217.___________0030_2 := false;
   AI_RAW_8217.PARAM_TYPE := 16#08;
   AI_RAW_8217.PARAM_RANGE := 16#17;
   AI_RAW_8217.PARAM_COEF := 16#02;
   AI_RAW_8217.___________0040_1 := false;
   AI_RAW_8217.___________0040_2 := false;
   AI_RAW_8217.VALUE_COEF := 0.003902;
   AI_RAW_8517.revInfo.REV_BLOCK := 'UT00801';
   AI_RAW_8517.revInfo.REV_NUMBER := '001.000';
   AI_RAW_8517.revInfo.REV_DATE := '2024-04-09';
   AI_RAW_8517.revInfo.REV_AUTHOR := 'M. Gledhill';
   AI_RAW_8517.___________0010_0 := false;
   AI_RAW_8517.___________0010_1 := false;
   AI_RAW_8517.AI_CODE := 16#8517;
   AI_RAW_8517.___________0020_0 := false;
   AI_RAW_8517.___________0020_1 := false;
   AI_RAW_8517.RAW_MIN := -12000;
   AI_RAW_8517.RAW_MAX := 13000;
   AI_RAW_8517.RAW_DESC := 'Thermal Resistance - 3-wire (Pt50 climate - 391)';
   AI_RAW_8517.___________0030_1 := false;
   AI_RAW_8517.___________0030_2 := false;
   AI_RAW_8517.PARAM_TYPE := 16#08;
   AI_RAW_8517.PARAM_RANGE := 16#17;
   AI_RAW_8517.PARAM_COEF := 16#05;
   AI_RAW_8517.___________0040_1 := false;
   AI_RAW_8517.___________0040_2 := false;
   AI_RAW_8517.VALUE_COEF := 0.00391;
   AI_RAW_8117.revInfo.REV_BLOCK := 'UT00801';
   AI_RAW_8117.revInfo.REV_NUMBER := '001.000';
   AI_RAW_8117.revInfo.REV_DATE := '2024-04-09';
   AI_RAW_8117.revInfo.REV_AUTHOR := 'M. Gledhill';
   AI_RAW_8117.___________0010_0 := false;
   AI_RAW_8117.___________0010_1 := false;
   AI_RAW_8117.AI_CODE := 16#8117;
   AI_RAW_8117.___________0020_0 := false;
   AI_RAW_8117.___________0020_1 := false;
   AI_RAW_8117.RAW_MIN := -12000;
   AI_RAW_8117.RAW_MAX := 13000;
   AI_RAW_8117.RAW_DESC := 'Thermal Resistance - 3-wire (Pt50 climate - 3916)';
   AI_RAW_8117.___________0030_1 := false;
   AI_RAW_8117.___________0030_2 := false;
   AI_RAW_8117.PARAM_TYPE := 16#08;
   AI_RAW_8117.PARAM_RANGE := 16#17;
   AI_RAW_8117.PARAM_COEF := 16#01;
   AI_RAW_8117.___________0040_1 := false;
   AI_RAW_8117.___________0040_2 := false;
   AI_RAW_8117.VALUE_COEF := 0.003916;
   AI_RAW_8317.revInfo.REV_BLOCK := 'UT00801';
   AI_RAW_8317.revInfo.REV_NUMBER := '001.000';
   AI_RAW_8317.revInfo.REV_DATE := '2024-04-09';
   AI_RAW_8317.revInfo.REV_AUTHOR := 'M. Gledhill';
   AI_RAW_8317.___________0010_0 := false;
   AI_RAW_8317.___________0010_1 := false;
   AI_RAW_8317.AI_CODE := 16#8317;
   AI_RAW_8317.___________0020_0 := false;
   AI_RAW_8317.___________0020_1 := false;
   AI_RAW_8317.RAW_MIN := -12000;
   AI_RAW_8317.RAW_MAX := 13000;
   AI_RAW_8317.RAW_DESC := 'Thermal Resistance - 3-wire (Pt50 climate - 392)';
   AI_RAW_8317.___________0030_1 := false;
   AI_RAW_8317.___________0030_2 := false;
   AI_RAW_8317.PARAM_TYPE := 16#08;
   AI_RAW_8317.PARAM_RANGE := 16#17;
   AI_RAW_8317.PARAM_COEF := 16#03;
   AI_RAW_8317.___________0040_1 := false;
   AI_RAW_8317.___________0040_2 := false;
   AI_RAW_8317.VALUE_COEF := 0.00392;
   AI_RAW_8016.revInfo.REV_BLOCK := 'UT00801';
   AI_RAW_8016.revInfo.REV_NUMBER := '001.000';
   AI_RAW_8016.revInfo.REV_DATE := '2024-04-09';
   AI_RAW_8016.revInfo.REV_AUTHOR := 'M. Gledhill';
   AI_RAW_8016.___________0010_0 := false;
   AI_RAW_8016.___________0010_1 := false;
   AI_RAW_8016.AI_CODE := 16#8016;
   AI_RAW_8016.___________0020_0 := false;
   AI_RAW_8016.___________0020_1 := false;
   AI_RAW_8016.RAW_MIN := -2000;
   AI_RAW_8016.RAW_MAX := 8500;
   AI_RAW_8016.RAW_DESC := 'Thermal Resistance - 3-wire (Pt50 standard - 3851)';
   AI_RAW_8016.___________0030_1 := false;
   AI_RAW_8016.___________0030_2 := false;
   AI_RAW_8016.PARAM_TYPE := 16#08;
   AI_RAW_8016.PARAM_RANGE := 16#16;
   AI_RAW_8016.PARAM_COEF := 16#00;
   AI_RAW_8016.___________0040_1 := false;
   AI_RAW_8016.___________0040_2 := false;
   AI_RAW_8016.VALUE_COEF := 0.003851;
   AI_RAW_8216.revInfo.REV_BLOCK := 'UT00801';
   AI_RAW_8216.revInfo.REV_NUMBER := '001.000';
   AI_RAW_8216.revInfo.REV_DATE := '2024-04-09';
   AI_RAW_8216.revInfo.REV_AUTHOR := 'M. Gledhill';
   AI_RAW_8216.___________0010_0 := false;
   AI_RAW_8216.___________0010_1 := false;
   AI_RAW_8216.AI_CODE := 16#8216;
   AI_RAW_8216.___________0020_0 := false;
   AI_RAW_8216.___________0020_1 := false;
   AI_RAW_8216.RAW_MIN := -2000;
   AI_RAW_8216.RAW_MAX := 8500;
   AI_RAW_8216.RAW_DESC := 'Thermal Resistance - 3-wire (Pt50 standard - 3902)';
   AI_RAW_8216.___________0030_1 := false;
   AI_RAW_8216.___________0030_2 := false;
   AI_RAW_8216.PARAM_TYPE := 16#08;
   AI_RAW_8216.PARAM_RANGE := 16#16;
   AI_RAW_8216.PARAM_COEF := 16#02;
   AI_RAW_8216.___________0040_1 := false;
   AI_RAW_8216.___________0040_2 := false;
   AI_RAW_8216.VALUE_COEF := 0.003902;
   AI_RAW_8516.revInfo.REV_BLOCK := 'UT00801';
   AI_RAW_8516.revInfo.REV_NUMBER := '001.000';
   AI_RAW_8516.revInfo.REV_DATE := '2024-04-09';
   AI_RAW_8516.revInfo.REV_AUTHOR := 'M. Gledhill';
   AI_RAW_8516.___________0010_0 := false;
   AI_RAW_8516.___________0010_1 := false;
   AI_RAW_8516.AI_CODE := 16#8516;
   AI_RAW_8516.___________0020_0 := false;
   AI_RAW_8516.___________0020_1 := false;
   AI_RAW_8516.RAW_MIN := -2000;
   AI_RAW_8516.RAW_MAX := 8500;
   AI_RAW_8516.RAW_DESC := 'Thermal Resistance - 3-wire (Pt50 standard - 391)';
   AI_RAW_8516.___________0030_1 := false;
   AI_RAW_8516.___________0030_2 := false;
   AI_RAW_8516.PARAM_TYPE := 16#08;
   AI_RAW_8516.PARAM_RANGE := 16#16;
   AI_RAW_8516.PARAM_COEF := 16#05;
   AI_RAW_8516.___________0040_1 := false;
   AI_RAW_8516.___________0040_2 := false;
   AI_RAW_8516.VALUE_COEF := 0.00391;
   AI_RAW_8116.revInfo.REV_BLOCK := 'UT00801';
   AI_RAW_8116.revInfo.REV_NUMBER := '001.000';
   AI_RAW_8116.revInfo.REV_DATE := '2024-04-09';
   AI_RAW_8116.revInfo.REV_AUTHOR := 'M. Gledhill';
   AI_RAW_8116.___________0010_0 := false;
   AI_RAW_8116.___________0010_1 := false;
   AI_RAW_8116.AI_CODE := 16#8116;
   AI_RAW_8116.___________0020_0 := false;
   AI_RAW_8116.___________0020_1 := false;
   AI_RAW_8116.RAW_MIN := -2000;
   AI_RAW_8116.RAW_MAX := 8500;
   AI_RAW_8116.RAW_DESC := 'Thermal Resistance - 3-wire (Pt50 standard - 3916)';
   AI_RAW_8116.___________0030_1 := false;
   AI_RAW_8116.___________0030_2 := false;
   AI_RAW_8116.PARAM_TYPE := 16#08;
   AI_RAW_8116.PARAM_RANGE := 16#16;
   AI_RAW_8116.PARAM_COEF := 16#01;
   AI_RAW_8116.___________0040_1 := false;
   AI_RAW_8116.___________0040_2 := false;
   AI_RAW_8116.VALUE_COEF := 0.003916;
   AI_RAW_8316.revInfo.REV_BLOCK := 'UT00801';
   AI_RAW_8316.revInfo.REV_NUMBER := '001.000';
   AI_RAW_8316.revInfo.REV_DATE := '2024-04-09';
   AI_RAW_8316.revInfo.REV_AUTHOR := 'M. Gledhill';
   AI_RAW_8316.___________0010_0 := false;
   AI_RAW_8316.___________0010_1 := false;
   AI_RAW_8316.AI_CODE := 16#8316;
   AI_RAW_8316.___________0020_0 := false;
   AI_RAW_8316.___________0020_1 := false;
   AI_RAW_8316.RAW_MIN := -2000;
   AI_RAW_8316.RAW_MAX := 8500;
   AI_RAW_8316.RAW_DESC := 'Thermal Resistance - 3-wire (Pt50 standard - 392)';
   AI_RAW_8316.___________0030_1 := false;
   AI_RAW_8316.___________0030_2 := false;
   AI_RAW_8316.PARAM_TYPE := 16#08;
   AI_RAW_8316.PARAM_RANGE := 16#16;
   AI_RAW_8316.PARAM_COEF := 16#03;
   AI_RAW_8316.___________0040_1 := false;
   AI_RAW_8316.___________0040_2 := false;
   AI_RAW_8316.VALUE_COEF := 0.00392;
   AI_RAW_8000.revInfo.REV_BLOCK := 'UT00801';
   AI_RAW_8000.revInfo.REV_NUMBER := '001.000';
   AI_RAW_8000.revInfo.REV_DATE := '2024-04-09';
   AI_RAW_8000.revInfo.REV_AUTHOR := 'M. Gledhill';
   AI_RAW_8000.___________0010_0 := false;
   AI_RAW_8000.___________0010_1 := false;
   AI_RAW_8000.AI_CODE := 16#8000;
   AI_RAW_8000.___________0020_0 := false;
   AI_RAW_8000.___________0020_1 := false;
   AI_RAW_8000.RAW_MIN := -12000;
   AI_RAW_8000.RAW_MAX := 13000;
   AI_RAW_8000.RAW_DESC := 'Thermal Resistance - 3-wire (Pt100 climate - 3851)';
   AI_RAW_8000.___________0030_1 := false;
   AI_RAW_8000.___________0030_2 := false;
   AI_RAW_8000.PARAM_TYPE := 16#08;
   AI_RAW_8000.PARAM_RANGE := 16#00;
   AI_RAW_8000.PARAM_COEF := 16#00;
   AI_RAW_8000.___________0040_1 := false;
   AI_RAW_8000.___________0040_2 := false;
   AI_RAW_8000.VALUE_COEF := 0.003851;
   AI_RAW_8200.revInfo.REV_BLOCK := 'UT00801';
   AI_RAW_8200.revInfo.REV_NUMBER := '001.000';
   AI_RAW_8200.revInfo.REV_DATE := '2024-04-09';
   AI_RAW_8200.revInfo.REV_AUTHOR := 'M. Gledhill';
   AI_RAW_8200.___________0010_0 := false;
   AI_RAW_8200.___________0010_1 := false;
   AI_RAW_8200.AI_CODE := 16#8200;
   AI_RAW_8200.___________0020_0 := false;
   AI_RAW_8200.___________0020_1 := false;
   AI_RAW_8200.RAW_MIN := -12000;
   AI_RAW_8200.RAW_MAX := 13000;
   AI_RAW_8200.RAW_DESC := 'Thermal Resistance - 3-wire (Pt100 climate - 3902)';
   AI_RAW_8200.___________0030_1 := false;
   AI_RAW_8200.___________0030_2 := false;
   AI_RAW_8200.PARAM_TYPE := 16#08;
   AI_RAW_8200.PARAM_RANGE := 16#00;
   AI_RAW_8200.PARAM_COEF := 16#02;
   AI_RAW_8200.___________0040_1 := false;
   AI_RAW_8200.___________0040_2 := false;
   AI_RAW_8200.VALUE_COEF := 0.003902;
   AI_RAW_8500.revInfo.REV_BLOCK := 'UT00801';
   AI_RAW_8500.revInfo.REV_NUMBER := '001.000';
   AI_RAW_8500.revInfo.REV_DATE := '2024-04-09';
   AI_RAW_8500.revInfo.REV_AUTHOR := 'M. Gledhill';
   AI_RAW_8500.___________0010_0 := false;
   AI_RAW_8500.___________0010_1 := false;
   AI_RAW_8500.AI_CODE := 16#8500;
   AI_RAW_8500.___________0020_0 := false;
   AI_RAW_8500.___________0020_1 := false;
   AI_RAW_8500.RAW_MIN := -12000;
   AI_RAW_8500.RAW_MAX := 13000;
   AI_RAW_8500.RAW_DESC := 'Thermal Resistance - 3-wire (Pt100 climate - 391)';
   AI_RAW_8500.___________0030_1 := false;
   AI_RAW_8500.___________0030_2 := false;
   AI_RAW_8500.PARAM_TYPE := 16#08;
   AI_RAW_8500.PARAM_RANGE := 16#00;
   AI_RAW_8500.PARAM_COEF := 16#05;
   AI_RAW_8500.___________0040_1 := false;
   AI_RAW_8500.___________0040_2 := false;
   AI_RAW_8500.VALUE_COEF := 0.00391;
   AI_RAW_8100.revInfo.REV_BLOCK := 'UT00801';
   AI_RAW_8100.revInfo.REV_NUMBER := '001.000';
   AI_RAW_8100.revInfo.REV_DATE := '2024-04-09';
   AI_RAW_8100.revInfo.REV_AUTHOR := 'M. Gledhill';
   AI_RAW_8100.___________0010_0 := false;
   AI_RAW_8100.___________0010_1 := false;
   AI_RAW_8100.AI_CODE := 16#8100;
   AI_RAW_8100.___________0020_0 := false;
   AI_RAW_8100.___________0020_1 := false;
   AI_RAW_8100.RAW_MIN := -12000;
   AI_RAW_8100.RAW_MAX := 13000;
   AI_RAW_8100.RAW_DESC := 'Thermal Resistance - 3-wire (Pt100 climate - 3916)';
   AI_RAW_8100.___________0030_1 := false;
   AI_RAW_8100.___________0030_2 := false;
   AI_RAW_8100.PARAM_TYPE := 16#08;
   AI_RAW_8100.PARAM_RANGE := 16#00;
   AI_RAW_8100.PARAM_COEF := 16#01;
   AI_RAW_8100.___________0040_1 := false;
   AI_RAW_8100.___________0040_2 := false;
   AI_RAW_8100.VALUE_COEF := 0.003916;
   AI_RAW_8300.revInfo.REV_BLOCK := 'UT00801';
   AI_RAW_8300.revInfo.REV_NUMBER := '001.000';
   AI_RAW_8300.revInfo.REV_DATE := '2024-04-09';
   AI_RAW_8300.revInfo.REV_AUTHOR := 'M. Gledhill';
   AI_RAW_8300.___________0010_0 := false;
   AI_RAW_8300.___________0010_1 := false;
   AI_RAW_8300.AI_CODE := 16#8300;
   AI_RAW_8300.___________0020_0 := false;
   AI_RAW_8300.___________0020_1 := false;
   AI_RAW_8300.RAW_MIN := -12000;
   AI_RAW_8300.RAW_MAX := 13000;
   AI_RAW_8300.RAW_DESC := 'Thermal Resistance - 3-wire (Pt100 climate - 392)';
   AI_RAW_8300.___________0030_1 := false;
   AI_RAW_8300.___________0030_2 := false;
   AI_RAW_8300.PARAM_TYPE := 16#08;
   AI_RAW_8300.PARAM_RANGE := 16#00;
   AI_RAW_8300.PARAM_COEF := 16#03;
   AI_RAW_8300.___________0040_1 := false;
   AI_RAW_8300.___________0040_2 := false;
   AI_RAW_8300.VALUE_COEF := 0.00392;
   AI_RAW_8002.revInfo.REV_BLOCK := 'UT00801';
   AI_RAW_8002.revInfo.REV_NUMBER := '001.000';
   AI_RAW_8002.revInfo.REV_DATE := '2024-04-09';
   AI_RAW_8002.revInfo.REV_AUTHOR := 'M. Gledhill';
   AI_RAW_8002.___________0010_0 := false;
   AI_RAW_8002.___________0010_1 := false;
   AI_RAW_8002.AI_CODE := 16#8002;
   AI_RAW_8002.___________0020_0 := false;
   AI_RAW_8002.___________0020_1 := false;
   AI_RAW_8002.RAW_MIN := -2000;
   AI_RAW_8002.RAW_MAX := 8500;
   AI_RAW_8002.RAW_DESC := 'Thermal Resistance - 3-wire (Pt100 standard - 3851)';
   AI_RAW_8002.___________0030_1 := false;
   AI_RAW_8002.___________0030_2 := false;
   AI_RAW_8002.PARAM_TYPE := 16#08;
   AI_RAW_8002.PARAM_RANGE := 16#02;
   AI_RAW_8002.PARAM_COEF := 16#00;
   AI_RAW_8002.___________0040_1 := false;
   AI_RAW_8002.___________0040_2 := false;
   AI_RAW_8002.VALUE_COEF := 0.003851;
   AI_RAW_8202.revInfo.REV_BLOCK := 'UT00801';
   AI_RAW_8202.revInfo.REV_NUMBER := '001.000';
   AI_RAW_8202.revInfo.REV_DATE := '2024-04-09';
   AI_RAW_8202.revInfo.REV_AUTHOR := 'M. Gledhill';
   AI_RAW_8202.___________0010_0 := false;
   AI_RAW_8202.___________0010_1 := false;
   AI_RAW_8202.AI_CODE := 16#8202;
   AI_RAW_8202.___________0020_0 := false;
   AI_RAW_8202.___________0020_1 := false;
   AI_RAW_8202.RAW_MIN := -2000;
   AI_RAW_8202.RAW_MAX := 8500;
   AI_RAW_8202.RAW_DESC := 'Thermal Resistance - 3-wire (Pt100 standard - 3902)';
   AI_RAW_8202.___________0030_1 := false;
   AI_RAW_8202.___________0030_2 := false;
   AI_RAW_8202.PARAM_TYPE := 16#08;
   AI_RAW_8202.PARAM_RANGE := 16#02;
   AI_RAW_8202.PARAM_COEF := 16#02;
   AI_RAW_8202.___________0040_1 := false;
   AI_RAW_8202.___________0040_2 := false;
   AI_RAW_8202.VALUE_COEF := 0.003902;
   AI_RAW_8502.revInfo.REV_BLOCK := 'UT00801';
   AI_RAW_8502.revInfo.REV_NUMBER := '001.000';
   AI_RAW_8502.revInfo.REV_DATE := '2024-04-09';
   AI_RAW_8502.revInfo.REV_AUTHOR := 'M. Gledhill';
   AI_RAW_8502.___________0010_0 := false;
   AI_RAW_8502.___________0010_1 := false;
   AI_RAW_8502.AI_CODE := 16#8502;
   AI_RAW_8502.___________0020_0 := false;
   AI_RAW_8502.___________0020_1 := false;
   AI_RAW_8502.RAW_MIN := -2000;
   AI_RAW_8502.RAW_MAX := 8500;
   AI_RAW_8502.RAW_DESC := 'Thermal Resistance - 3-wire (Pt100 standard - 391)';
   AI_RAW_8502.___________0030_1 := false;
   AI_RAW_8502.___________0030_2 := false;
   AI_RAW_8502.PARAM_TYPE := 16#08;
   AI_RAW_8502.PARAM_RANGE := 16#02;
   AI_RAW_8502.PARAM_COEF := 16#05;
   AI_RAW_8502.___________0040_1 := false;
   AI_RAW_8502.___________0040_2 := false;
   AI_RAW_8502.VALUE_COEF := 0.00391;
   AI_RAW_8102.revInfo.REV_BLOCK := 'UT00801';
   AI_RAW_8102.revInfo.REV_NUMBER := '001.000';
   AI_RAW_8102.revInfo.REV_DATE := '2024-04-09';
   AI_RAW_8102.revInfo.REV_AUTHOR := 'M. Gledhill';
   AI_RAW_8102.___________0010_0 := false;
   AI_RAW_8102.___________0010_1 := false;
   AI_RAW_8102.AI_CODE := 16#8102;
   AI_RAW_8102.___________0020_0 := false;
   AI_RAW_8102.___________0020_1 := false;
   AI_RAW_8102.RAW_MIN := -2000;
   AI_RAW_8102.RAW_MAX := 8500;
   AI_RAW_8102.RAW_DESC := 'Thermal Resistance - 3-wire (Pt100 standard - 3916)';
   AI_RAW_8102.___________0030_1 := false;
   AI_RAW_8102.___________0030_2 := false;
   AI_RAW_8102.PARAM_TYPE := 16#08;
   AI_RAW_8102.PARAM_RANGE := 16#02;
   AI_RAW_8102.PARAM_COEF := 16#01;
   AI_RAW_8102.___________0040_1 := false;
   AI_RAW_8102.___________0040_2 := false;
   AI_RAW_8102.VALUE_COEF := 0.003916;
   AI_RAW_8302.revInfo.REV_BLOCK := 'UT00801';
   AI_RAW_8302.revInfo.REV_NUMBER := '001.000';
   AI_RAW_8302.revInfo.REV_DATE := '2024-04-09';
   AI_RAW_8302.revInfo.REV_AUTHOR := 'M. Gledhill';
   AI_RAW_8302.___________0010_0 := false;
   AI_RAW_8302.___________0010_1 := false;
   AI_RAW_8302.AI_CODE := 16#8302;
   AI_RAW_8302.___________0020_0 := false;
   AI_RAW_8302.___________0020_1 := false;
   AI_RAW_8302.RAW_MIN := -2000;
   AI_RAW_8302.RAW_MAX := 8500;
   AI_RAW_8302.RAW_DESC := 'Thermal Resistance - 3-wire (Pt100 standard - 392)';
   AI_RAW_8302.___________0030_1 := false;
   AI_RAW_8302.___________0030_2 := false;
   AI_RAW_8302.PARAM_TYPE := 16#08;
   AI_RAW_8302.PARAM_RANGE := 16#02;
   AI_RAW_8302.PARAM_COEF := 16#03;
   AI_RAW_8302.___________0040_1 := false;
   AI_RAW_8302.___________0040_2 := false;
   AI_RAW_8302.VALUE_COEF := 0.00392;
   AI_RAW_8007.revInfo.REV_BLOCK := 'UT00801';
   AI_RAW_8007.revInfo.REV_NUMBER := '001.000';
   AI_RAW_8007.revInfo.REV_DATE := '2024-04-09';
   AI_RAW_8007.revInfo.REV_AUTHOR := 'M. Gledhill';
   AI_RAW_8007.___________0010_0 := false;
   AI_RAW_8007.___________0010_1 := false;
   AI_RAW_8007.AI_CODE := 16#8007;
   AI_RAW_8007.___________0020_0 := false;
   AI_RAW_8007.___________0020_1 := false;
   AI_RAW_8007.RAW_MIN := -12000;
   AI_RAW_8007.RAW_MAX := 13000;
   AI_RAW_8007.RAW_DESC := 'Thermal Resistance - 3-wire (Pt200 climate - 3851)';
   AI_RAW_8007.___________0030_1 := false;
   AI_RAW_8007.___________0030_2 := false;
   AI_RAW_8007.PARAM_TYPE := 16#08;
   AI_RAW_8007.PARAM_RANGE := 16#07;
   AI_RAW_8007.PARAM_COEF := 16#00;
   AI_RAW_8007.___________0040_1 := false;
   AI_RAW_8007.___________0040_2 := false;
   AI_RAW_8007.VALUE_COEF := 0.003851;
   AI_RAW_8207.revInfo.REV_BLOCK := 'UT00801';
   AI_RAW_8207.revInfo.REV_NUMBER := '001.000';
   AI_RAW_8207.revInfo.REV_DATE := '2024-04-09';
   AI_RAW_8207.revInfo.REV_AUTHOR := 'M. Gledhill';
   AI_RAW_8207.___________0010_0 := false;
   AI_RAW_8207.___________0010_1 := false;
   AI_RAW_8207.AI_CODE := 16#8207;
   AI_RAW_8207.___________0020_0 := false;
   AI_RAW_8207.___________0020_1 := false;
   AI_RAW_8207.RAW_MIN := -12000;
   AI_RAW_8207.RAW_MAX := 13000;
   AI_RAW_8207.RAW_DESC := 'Thermal Resistance - 3-wire (Pt200 climate - 3902)';
   AI_RAW_8207.___________0030_1 := false;
   AI_RAW_8207.___________0030_2 := false;
   AI_RAW_8207.PARAM_TYPE := 16#08;
   AI_RAW_8207.PARAM_RANGE := 16#07;
   AI_RAW_8207.PARAM_COEF := 16#02;
   AI_RAW_8207.___________0040_1 := false;
   AI_RAW_8207.___________0040_2 := false;
   AI_RAW_8207.VALUE_COEF := 0.003902;
   AI_RAW_8507.revInfo.REV_BLOCK := 'UT00801';
   AI_RAW_8507.revInfo.REV_NUMBER := '001.000';
   AI_RAW_8507.revInfo.REV_DATE := '2024-04-09';
   AI_RAW_8507.revInfo.REV_AUTHOR := 'M. Gledhill';
   AI_RAW_8507.___________0010_0 := false;
   AI_RAW_8507.___________0010_1 := false;
   AI_RAW_8507.AI_CODE := 16#8507;
   AI_RAW_8507.___________0020_0 := false;
   AI_RAW_8507.___________0020_1 := false;
   AI_RAW_8507.RAW_MIN := -12000;
   AI_RAW_8507.RAW_MAX := 13000;
   AI_RAW_8507.RAW_DESC := 'Thermal Resistance - 3-wire (Pt200 climate - 391)';
   AI_RAW_8507.___________0030_1 := false;
   AI_RAW_8507.___________0030_2 := false;
   AI_RAW_8507.PARAM_TYPE := 16#08;
   AI_RAW_8507.PARAM_RANGE := 16#07;
   AI_RAW_8507.PARAM_COEF := 16#05;
   AI_RAW_8507.___________0040_1 := false;
   AI_RAW_8507.___________0040_2 := false;
   AI_RAW_8507.VALUE_COEF := 0.00391;
   AI_RAW_8107.revInfo.REV_BLOCK := 'UT00801';
   AI_RAW_8107.revInfo.REV_NUMBER := '001.000';
   AI_RAW_8107.revInfo.REV_DATE := '2024-04-09';
   AI_RAW_8107.revInfo.REV_AUTHOR := 'M. Gledhill';
   AI_RAW_8107.___________0010_0 := false;
   AI_RAW_8107.___________0010_1 := false;
   AI_RAW_8107.AI_CODE := 16#8107;
   AI_RAW_8107.___________0020_0 := false;
   AI_RAW_8107.___________0020_1 := false;
   AI_RAW_8107.RAW_MIN := -12000;
   AI_RAW_8107.RAW_MAX := 13000;
   AI_RAW_8107.RAW_DESC := 'Thermal Resistance - 3-wire (Pt200 climate - 3916)';
   AI_RAW_8107.___________0030_1 := false;
   AI_RAW_8107.___________0030_2 := false;
   AI_RAW_8107.PARAM_TYPE := 16#08;
   AI_RAW_8107.PARAM_RANGE := 16#07;
   AI_RAW_8107.PARAM_COEF := 16#01;
   AI_RAW_8107.___________0040_1 := false;
   AI_RAW_8107.___________0040_2 := false;
   AI_RAW_8107.VALUE_COEF := 0.003916;
   AI_RAW_8307.revInfo.REV_BLOCK := 'UT00801';
   AI_RAW_8307.revInfo.REV_NUMBER := '001.000';
   AI_RAW_8307.revInfo.REV_DATE := '2024-04-09';
   AI_RAW_8307.revInfo.REV_AUTHOR := 'M. Gledhill';
   AI_RAW_8307.___________0010_0 := false;
   AI_RAW_8307.___________0010_1 := false;
   AI_RAW_8307.AI_CODE := 16#8307;
   AI_RAW_8307.___________0020_0 := false;
   AI_RAW_8307.___________0020_1 := false;
   AI_RAW_8307.RAW_MIN := -12000;
   AI_RAW_8307.RAW_MAX := 13000;
   AI_RAW_8307.RAW_DESC := 'Thermal Resistance - 3-wire (Pt200 climate - 392)';
   AI_RAW_8307.___________0030_1 := false;
   AI_RAW_8307.___________0030_2 := false;
   AI_RAW_8307.PARAM_TYPE := 16#08;
   AI_RAW_8307.PARAM_RANGE := 16#07;
   AI_RAW_8307.PARAM_COEF := 16#03;
   AI_RAW_8307.___________0040_1 := false;
   AI_RAW_8307.___________0040_2 := false;
   AI_RAW_8307.VALUE_COEF := 0.00392;
   AI_RAW_800B.revInfo.REV_BLOCK := 'UT00801';
   AI_RAW_800B.revInfo.REV_NUMBER := '001.000';
   AI_RAW_800B.revInfo.REV_DATE := '2024-04-09';
   AI_RAW_800B.revInfo.REV_AUTHOR := 'M. Gledhill';
   AI_RAW_800B.___________0010_0 := false;
   AI_RAW_800B.___________0010_1 := false;
   AI_RAW_800B.AI_CODE := 16#800B;
   AI_RAW_800B.___________0020_0 := false;
   AI_RAW_800B.___________0020_1 := false;
   AI_RAW_800B.RAW_MIN := -2000;
   AI_RAW_800B.RAW_MAX := 8500;
   AI_RAW_800B.RAW_DESC := 'Thermal Resistance - 3-wire (Pt200 standard - 3851)';
   AI_RAW_800B.___________0030_1 := false;
   AI_RAW_800B.___________0030_2 := false;
   AI_RAW_800B.PARAM_TYPE := 16#08;
   AI_RAW_800B.PARAM_RANGE := 16#0B;
   AI_RAW_800B.PARAM_COEF := 16#00;
   AI_RAW_800B.___________0040_1 := false;
   AI_RAW_800B.___________0040_2 := false;
   AI_RAW_800B.VALUE_COEF := 0.003851;
   AI_RAW_820B.revInfo.REV_BLOCK := 'UT00801';
   AI_RAW_820B.revInfo.REV_NUMBER := '001.000';
   AI_RAW_820B.revInfo.REV_DATE := '2024-04-09';
   AI_RAW_820B.revInfo.REV_AUTHOR := 'M. Gledhill';
   AI_RAW_820B.___________0010_0 := false;
   AI_RAW_820B.___________0010_1 := false;
   AI_RAW_820B.AI_CODE := 16#820B;
   AI_RAW_820B.___________0020_0 := false;
   AI_RAW_820B.___________0020_1 := false;
   AI_RAW_820B.RAW_MIN := -2000;
   AI_RAW_820B.RAW_MAX := 8500;
   AI_RAW_820B.RAW_DESC := 'Thermal Resistance - 3-wire (Pt200 standard - 3902)';
   AI_RAW_820B.___________0030_1 := false;
   AI_RAW_820B.___________0030_2 := false;
   AI_RAW_820B.PARAM_TYPE := 16#08;
   AI_RAW_820B.PARAM_RANGE := 16#0B;
   AI_RAW_820B.PARAM_COEF := 16#02;
   AI_RAW_820B.___________0040_1 := false;
   AI_RAW_820B.___________0040_2 := false;
   AI_RAW_820B.VALUE_COEF := 0.003902;
   AI_RAW_850B.revInfo.REV_BLOCK := 'UT00801';
   AI_RAW_850B.revInfo.REV_NUMBER := '001.000';
   AI_RAW_850B.revInfo.REV_DATE := '2024-04-09';
   AI_RAW_850B.revInfo.REV_AUTHOR := 'M. Gledhill';
   AI_RAW_850B.___________0010_0 := false;
   AI_RAW_850B.___________0010_1 := false;
   AI_RAW_850B.AI_CODE := 16#850B;
   AI_RAW_850B.___________0020_0 := false;
   AI_RAW_850B.___________0020_1 := false;
   AI_RAW_850B.RAW_MIN := -2000;
   AI_RAW_850B.RAW_MAX := 8500;
   AI_RAW_850B.RAW_DESC := 'Thermal Resistance - 3-wire (Pt200 standard - 391)';
   AI_RAW_850B.___________0030_1 := false;
   AI_RAW_850B.___________0030_2 := false;
   AI_RAW_850B.PARAM_TYPE := 16#08;
   AI_RAW_850B.PARAM_RANGE := 16#0B;
   AI_RAW_850B.PARAM_COEF := 16#05;
   AI_RAW_850B.___________0040_1 := false;
   AI_RAW_850B.___________0040_2 := false;
   AI_RAW_850B.VALUE_COEF := 0.00391;
   AI_RAW_810B.revInfo.REV_BLOCK := 'UT00801';
   AI_RAW_810B.revInfo.REV_NUMBER := '001.000';
   AI_RAW_810B.revInfo.REV_DATE := '2024-04-09';
   AI_RAW_810B.revInfo.REV_AUTHOR := 'M. Gledhill';
   AI_RAW_810B.___________0010_0 := false;
   AI_RAW_810B.___________0010_1 := false;
   AI_RAW_810B.AI_CODE := 16#810B;
   AI_RAW_810B.___________0020_0 := false;
   AI_RAW_810B.___________0020_1 := false;
   AI_RAW_810B.RAW_MIN := -2000;
   AI_RAW_810B.RAW_MAX := 8500;
   AI_RAW_810B.RAW_DESC := 'Thermal Resistance - 3-wire (Pt200 standard - 3916)';
   AI_RAW_810B.___________0030_1 := false;
   AI_RAW_810B.___________0030_2 := false;
   AI_RAW_810B.PARAM_TYPE := 16#08;
   AI_RAW_810B.PARAM_RANGE := 16#0B;
   AI_RAW_810B.PARAM_COEF := 16#01;
   AI_RAW_810B.___________0040_1 := false;
   AI_RAW_810B.___________0040_2 := false;
   AI_RAW_810B.VALUE_COEF := 0.003916;
   AI_RAW_830B.revInfo.REV_BLOCK := 'UT00801';
   AI_RAW_830B.revInfo.REV_NUMBER := '001.000';
   AI_RAW_830B.revInfo.REV_DATE := '2024-04-09';
   AI_RAW_830B.revInfo.REV_AUTHOR := 'M. Gledhill';
   AI_RAW_830B.___________0010_0 := false;
   AI_RAW_830B.___________0010_1 := false;
   AI_RAW_830B.AI_CODE := 16#830B;
   AI_RAW_830B.___________0020_0 := false;
   AI_RAW_830B.___________0020_1 := false;
   AI_RAW_830B.RAW_MIN := -2000;
   AI_RAW_830B.RAW_MAX := 8500;
   AI_RAW_830B.RAW_DESC := 'Thermal Resistance - 3-wire (Pt200 standard - 392)';
   AI_RAW_830B.___________0030_1 := false;
   AI_RAW_830B.___________0030_2 := false;
   AI_RAW_830B.PARAM_TYPE := 16#08;
   AI_RAW_830B.PARAM_RANGE := 16#0B;
   AI_RAW_830B.PARAM_COEF := 16#03;
   AI_RAW_830B.___________0040_1 := false;
   AI_RAW_830B.___________0040_2 := false;
   AI_RAW_830B.VALUE_COEF := 0.00392;
   AI_RAW_8008.revInfo.REV_BLOCK := 'UT00801';
   AI_RAW_8008.revInfo.REV_NUMBER := '001.000';
   AI_RAW_8008.revInfo.REV_DATE := '2024-04-09';
   AI_RAW_8008.revInfo.REV_AUTHOR := 'M. Gledhill';
   AI_RAW_8008.___________0010_0 := false;
   AI_RAW_8008.___________0010_1 := false;
   AI_RAW_8008.AI_CODE := 16#8008;
   AI_RAW_8008.___________0020_0 := false;
   AI_RAW_8008.___________0020_1 := false;
   AI_RAW_8008.RAW_MIN := -12000;
   AI_RAW_8008.RAW_MAX := 13000;
   AI_RAW_8008.RAW_DESC := 'Thermal Resistance - 3-wire (Pt500 climate - 3851)';
   AI_RAW_8008.___________0030_1 := false;
   AI_RAW_8008.___________0030_2 := false;
   AI_RAW_8008.PARAM_TYPE := 16#08;
   AI_RAW_8008.PARAM_RANGE := 16#08;
   AI_RAW_8008.PARAM_COEF := 16#00;
   AI_RAW_8008.___________0040_1 := false;
   AI_RAW_8008.___________0040_2 := false;
   AI_RAW_8008.VALUE_COEF := 0.003851;
   AI_RAW_8208.revInfo.REV_BLOCK := 'UT00801';
   AI_RAW_8208.revInfo.REV_NUMBER := '001.000';
   AI_RAW_8208.revInfo.REV_DATE := '2024-04-09';
   AI_RAW_8208.revInfo.REV_AUTHOR := 'M. Gledhill';
   AI_RAW_8208.___________0010_0 := false;
   AI_RAW_8208.___________0010_1 := false;
   AI_RAW_8208.AI_CODE := 16#8208;
   AI_RAW_8208.___________0020_0 := false;
   AI_RAW_8208.___________0020_1 := false;
   AI_RAW_8208.RAW_MIN := -12000;
   AI_RAW_8208.RAW_MAX := 13000;
   AI_RAW_8208.RAW_DESC := 'Thermal Resistance - 3-wire (Pt500 climate - 3902)';
   AI_RAW_8208.___________0030_1 := false;
   AI_RAW_8208.___________0030_2 := false;
   AI_RAW_8208.PARAM_TYPE := 16#08;
   AI_RAW_8208.PARAM_RANGE := 16#08;
   AI_RAW_8208.PARAM_COEF := 16#02;
   AI_RAW_8208.___________0040_1 := false;
   AI_RAW_8208.___________0040_2 := false;
   AI_RAW_8208.VALUE_COEF := 0.003902;
   AI_RAW_8508.revInfo.REV_BLOCK := 'UT00801';
   AI_RAW_8508.revInfo.REV_NUMBER := '001.000';
   AI_RAW_8508.revInfo.REV_DATE := '2024-04-09';
   AI_RAW_8508.revInfo.REV_AUTHOR := 'M. Gledhill';
   AI_RAW_8508.___________0010_0 := false;
   AI_RAW_8508.___________0010_1 := false;
   AI_RAW_8508.AI_CODE := 16#8508;
   AI_RAW_8508.___________0020_0 := false;
   AI_RAW_8508.___________0020_1 := false;
   AI_RAW_8508.RAW_MIN := -12000;
   AI_RAW_8508.RAW_MAX := 13000;
   AI_RAW_8508.RAW_DESC := 'Thermal Resistance - 3-wire (Pt500 climate - 391)';
   AI_RAW_8508.___________0030_1 := false;
   AI_RAW_8508.___________0030_2 := false;
   AI_RAW_8508.PARAM_TYPE := 16#08;
   AI_RAW_8508.PARAM_RANGE := 16#08;
   AI_RAW_8508.PARAM_COEF := 16#05;
   AI_RAW_8508.___________0040_1 := false;
   AI_RAW_8508.___________0040_2 := false;
   AI_RAW_8508.VALUE_COEF := 0.00391;
   AI_RAW_8108.revInfo.REV_BLOCK := 'UT00801';
   AI_RAW_8108.revInfo.REV_NUMBER := '001.000';
   AI_RAW_8108.revInfo.REV_DATE := '2024-04-09';
   AI_RAW_8108.revInfo.REV_AUTHOR := 'M. Gledhill';
   AI_RAW_8108.___________0010_0 := false;
   AI_RAW_8108.___________0010_1 := false;
   AI_RAW_8108.AI_CODE := 16#8108;
   AI_RAW_8108.___________0020_0 := false;
   AI_RAW_8108.___________0020_1 := false;
   AI_RAW_8108.RAW_MIN := -12000;
   AI_RAW_8108.RAW_MAX := 13000;
   AI_RAW_8108.RAW_DESC := 'Thermal Resistance - 3-wire (Pt500 climate - 3916)';
   AI_RAW_8108.___________0030_1 := false;
   AI_RAW_8108.___________0030_2 := false;
   AI_RAW_8108.PARAM_TYPE := 16#08;
   AI_RAW_8108.PARAM_RANGE := 16#08;
   AI_RAW_8108.PARAM_COEF := 16#01;
   AI_RAW_8108.___________0040_1 := false;
   AI_RAW_8108.___________0040_2 := false;
   AI_RAW_8108.VALUE_COEF := 0.003916;
   AI_RAW_8308.revInfo.REV_BLOCK := 'UT00801';
   AI_RAW_8308.revInfo.REV_NUMBER := '001.000';
   AI_RAW_8308.revInfo.REV_DATE := '2024-04-09';
   AI_RAW_8308.revInfo.REV_AUTHOR := 'M. Gledhill';
   AI_RAW_8308.___________0010_0 := false;
   AI_RAW_8308.___________0010_1 := false;
   AI_RAW_8308.AI_CODE := 16#8308;
   AI_RAW_8308.___________0020_0 := false;
   AI_RAW_8308.___________0020_1 := false;
   AI_RAW_8308.RAW_MIN := -12000;
   AI_RAW_8308.RAW_MAX := 13000;
   AI_RAW_8308.RAW_DESC := 'Thermal Resistance - 3-wire (Pt500 climate - 392)';
   AI_RAW_8308.___________0030_1 := false;
   AI_RAW_8308.___________0030_2 := false;
   AI_RAW_8308.PARAM_TYPE := 16#08;
   AI_RAW_8308.PARAM_RANGE := 16#08;
   AI_RAW_8308.PARAM_COEF := 16#03;
   AI_RAW_8308.___________0040_1 := false;
   AI_RAW_8308.___________0040_2 := false;
   AI_RAW_8308.VALUE_COEF := 0.00392;
   AI_RAW_8004.revInfo.REV_BLOCK := 'UT00801';
   AI_RAW_8004.revInfo.REV_NUMBER := '001.000';
   AI_RAW_8004.revInfo.REV_DATE := '2024-04-09';
   AI_RAW_8004.revInfo.REV_AUTHOR := 'M. Gledhill';
   AI_RAW_8004.___________0010_0 := false;
   AI_RAW_8004.___________0010_1 := false;
   AI_RAW_8004.AI_CODE := 16#8004;
   AI_RAW_8004.___________0020_0 := false;
   AI_RAW_8004.___________0020_1 := false;
   AI_RAW_8004.RAW_MIN := -2000;
   AI_RAW_8004.RAW_MAX := 8500;
   AI_RAW_8004.RAW_DESC := 'Thermal Resistance - 3-wire (Pt500 standard - 3851)';
   AI_RAW_8004.___________0030_1 := false;
   AI_RAW_8004.___________0030_2 := false;
   AI_RAW_8004.PARAM_TYPE := 16#08;
   AI_RAW_8004.PARAM_RANGE := 16#04;
   AI_RAW_8004.PARAM_COEF := 16#00;
   AI_RAW_8004.___________0040_1 := false;
   AI_RAW_8004.___________0040_2 := false;
   AI_RAW_8004.VALUE_COEF := 0.003851;
   AI_RAW_8204.revInfo.REV_BLOCK := 'UT00801';
   AI_RAW_8204.revInfo.REV_NUMBER := '001.000';
   AI_RAW_8204.revInfo.REV_DATE := '2024-04-09';
   AI_RAW_8204.revInfo.REV_AUTHOR := 'M. Gledhill';
   AI_RAW_8204.___________0010_0 := false;
   AI_RAW_8204.___________0010_1 := false;
   AI_RAW_8204.AI_CODE := 16#8204;
   AI_RAW_8204.___________0020_0 := false;
   AI_RAW_8204.___________0020_1 := false;
   AI_RAW_8204.RAW_MIN := -2000;
   AI_RAW_8204.RAW_MAX := 8500;
   AI_RAW_8204.RAW_DESC := 'Thermal Resistance - 3-wire (Pt500 standard - 3902)';
   AI_RAW_8204.___________0030_1 := false;
   AI_RAW_8204.___________0030_2 := false;
   AI_RAW_8204.PARAM_TYPE := 16#08;
   AI_RAW_8204.PARAM_RANGE := 16#04;
   AI_RAW_8204.PARAM_COEF := 16#02;
   AI_RAW_8204.___________0040_1 := false;
   AI_RAW_8204.___________0040_2 := false;
   AI_RAW_8204.VALUE_COEF := 0.003902;
   AI_RAW_8504.revInfo.REV_BLOCK := 'UT00801';
   AI_RAW_8504.revInfo.REV_NUMBER := '001.000';
   AI_RAW_8504.revInfo.REV_DATE := '2024-04-09';
   AI_RAW_8504.revInfo.REV_AUTHOR := 'M. Gledhill';
   AI_RAW_8504.___________0010_0 := false;
   AI_RAW_8504.___________0010_1 := false;
   AI_RAW_8504.AI_CODE := 16#8504;
   AI_RAW_8504.___________0020_0 := false;
   AI_RAW_8504.___________0020_1 := false;
   AI_RAW_8504.RAW_MIN := -2000;
   AI_RAW_8504.RAW_MAX := 8500;
   AI_RAW_8504.RAW_DESC := 'Thermal Resistance - 3-wire (Pt500 standard - 391)';
   AI_RAW_8504.___________0030_1 := false;
   AI_RAW_8504.___________0030_2 := false;
   AI_RAW_8504.PARAM_TYPE := 16#08;
   AI_RAW_8504.PARAM_RANGE := 16#04;
   AI_RAW_8504.PARAM_COEF := 16#05;
   AI_RAW_8504.___________0040_1 := false;
   AI_RAW_8504.___________0040_2 := false;
   AI_RAW_8504.VALUE_COEF := 0.00391;
   AI_RAW_8104.revInfo.REV_BLOCK := 'UT00801';
   AI_RAW_8104.revInfo.REV_NUMBER := '001.000';
   AI_RAW_8104.revInfo.REV_DATE := '2024-04-09';
   AI_RAW_8104.revInfo.REV_AUTHOR := 'M. Gledhill';
   AI_RAW_8104.___________0010_0 := false;
   AI_RAW_8104.___________0010_1 := false;
   AI_RAW_8104.AI_CODE := 16#8104;
   AI_RAW_8104.___________0020_0 := false;
   AI_RAW_8104.___________0020_1 := false;
   AI_RAW_8104.RAW_MIN := -2000;
   AI_RAW_8104.RAW_MAX := 8500;
   AI_RAW_8104.RAW_DESC := 'Thermal Resistance - 3-wire (Pt500 standard - 3916)';
   AI_RAW_8104.___________0030_1 := false;
   AI_RAW_8104.___________0030_2 := false;
   AI_RAW_8104.PARAM_TYPE := 16#08;
   AI_RAW_8104.PARAM_RANGE := 16#04;
   AI_RAW_8104.PARAM_COEF := 16#01;
   AI_RAW_8104.___________0040_1 := false;
   AI_RAW_8104.___________0040_2 := false;
   AI_RAW_8104.VALUE_COEF := 0.003916;
   AI_RAW_8304.revInfo.REV_BLOCK := 'UT00801';
   AI_RAW_8304.revInfo.REV_NUMBER := '001.000';
   AI_RAW_8304.revInfo.REV_DATE := '2024-04-09';
   AI_RAW_8304.revInfo.REV_AUTHOR := 'M. Gledhill';
   AI_RAW_8304.___________0010_0 := false;
   AI_RAW_8304.___________0010_1 := false;
   AI_RAW_8304.AI_CODE := 16#8304;
   AI_RAW_8304.___________0020_0 := false;
   AI_RAW_8304.___________0020_1 := false;
   AI_RAW_8304.RAW_MIN := -2000;
   AI_RAW_8304.RAW_MAX := 8500;
   AI_RAW_8304.RAW_DESC := 'Thermal Resistance - 3-wire (Pt500 standard - 392)';
   AI_RAW_8304.___________0030_1 := false;
   AI_RAW_8304.___________0030_2 := false;
   AI_RAW_8304.PARAM_TYPE := 16#08;
   AI_RAW_8304.PARAM_RANGE := 16#04;
   AI_RAW_8304.PARAM_COEF := 16#03;
   AI_RAW_8304.___________0040_1 := false;
   AI_RAW_8304.___________0040_2 := false;
   AI_RAW_8304.VALUE_COEF := 0.00392;
   AI_RAW_8009.revInfo.REV_BLOCK := 'UT00801';
   AI_RAW_8009.revInfo.REV_NUMBER := '001.000';
   AI_RAW_8009.revInfo.REV_DATE := '2024-04-09';
   AI_RAW_8009.revInfo.REV_AUTHOR := 'M. Gledhill';
   AI_RAW_8009.___________0010_0 := false;
   AI_RAW_8009.___________0010_1 := false;
   AI_RAW_8009.AI_CODE := 16#8009;
   AI_RAW_8009.___________0020_0 := false;
   AI_RAW_8009.___________0020_1 := false;
   AI_RAW_8009.RAW_MIN := -12000;
   AI_RAW_8009.RAW_MAX := 13000;
   AI_RAW_8009.RAW_DESC := 'Thermal Resistance - 3-wire (Pt1000 climate - 3851)';
   AI_RAW_8009.___________0030_1 := false;
   AI_RAW_8009.___________0030_2 := false;
   AI_RAW_8009.PARAM_TYPE := 16#08;
   AI_RAW_8009.PARAM_RANGE := 16#09;
   AI_RAW_8009.PARAM_COEF := 16#00;
   AI_RAW_8009.___________0040_1 := false;
   AI_RAW_8009.___________0040_2 := false;
   AI_RAW_8009.VALUE_COEF := 0.003851;
   AI_RAW_8209.revInfo.REV_BLOCK := 'UT00801';
   AI_RAW_8209.revInfo.REV_NUMBER := '001.000';
   AI_RAW_8209.revInfo.REV_DATE := '2024-04-09';
   AI_RAW_8209.revInfo.REV_AUTHOR := 'M. Gledhill';
   AI_RAW_8209.___________0010_0 := false;
   AI_RAW_8209.___________0010_1 := false;
   AI_RAW_8209.AI_CODE := 16#8209;
   AI_RAW_8209.___________0020_0 := false;
   AI_RAW_8209.___________0020_1 := false;
   AI_RAW_8209.RAW_MIN := -12000;
   AI_RAW_8209.RAW_MAX := 13000;
   AI_RAW_8209.RAW_DESC := 'Thermal Resistance - 3-wire (Pt1000 climate - 3902)';
   AI_RAW_8209.___________0030_1 := false;
   AI_RAW_8209.___________0030_2 := false;
   AI_RAW_8209.PARAM_TYPE := 16#08;
   AI_RAW_8209.PARAM_RANGE := 16#09;
   AI_RAW_8209.PARAM_COEF := 16#02;
   AI_RAW_8209.___________0040_1 := false;
   AI_RAW_8209.___________0040_2 := false;
   AI_RAW_8209.VALUE_COEF := 0.003902;
   AI_RAW_8509.revInfo.REV_BLOCK := 'UT00801';
   AI_RAW_8509.revInfo.REV_NUMBER := '001.000';
   AI_RAW_8509.revInfo.REV_DATE := '2024-04-09';
   AI_RAW_8509.revInfo.REV_AUTHOR := 'M. Gledhill';
   AI_RAW_8509.___________0010_0 := false;
   AI_RAW_8509.___________0010_1 := false;
   AI_RAW_8509.AI_CODE := 16#8509;
   AI_RAW_8509.___________0020_0 := false;
   AI_RAW_8509.___________0020_1 := false;
   AI_RAW_8509.RAW_MIN := -12000;
   AI_RAW_8509.RAW_MAX := 13000;
   AI_RAW_8509.RAW_DESC := 'Thermal Resistance - 3-wire (Pt1000 climate - 391)';
   AI_RAW_8509.___________0030_1 := false;
   AI_RAW_8509.___________0030_2 := false;
   AI_RAW_8509.PARAM_TYPE := 16#08;
   AI_RAW_8509.PARAM_RANGE := 16#09;
   AI_RAW_8509.PARAM_COEF := 16#05;
   AI_RAW_8509.___________0040_1 := false;
   AI_RAW_8509.___________0040_2 := false;
   AI_RAW_8509.VALUE_COEF := 0.00391;
   AI_RAW_8109.revInfo.REV_BLOCK := 'UT00801';
   AI_RAW_8109.revInfo.REV_NUMBER := '001.000';
   AI_RAW_8109.revInfo.REV_DATE := '2024-04-09';
   AI_RAW_8109.revInfo.REV_AUTHOR := 'M. Gledhill';
   AI_RAW_8109.___________0010_0 := false;
   AI_RAW_8109.___________0010_1 := false;
   AI_RAW_8109.AI_CODE := 16#8109;
   AI_RAW_8109.___________0020_0 := false;
   AI_RAW_8109.___________0020_1 := false;
   AI_RAW_8109.RAW_MIN := -12000;
   AI_RAW_8109.RAW_MAX := 13000;
   AI_RAW_8109.RAW_DESC := 'Thermal Resistance - 3-wire (Pt1000 climate - 3916)';
   AI_RAW_8109.___________0030_1 := false;
   AI_RAW_8109.___________0030_2 := false;
   AI_RAW_8109.PARAM_TYPE := 16#08;
   AI_RAW_8109.PARAM_RANGE := 16#09;
   AI_RAW_8109.PARAM_COEF := 16#01;
   AI_RAW_8109.___________0040_1 := false;
   AI_RAW_8109.___________0040_2 := false;
   AI_RAW_8109.VALUE_COEF := 0.003916;
   AI_RAW_8309.revInfo.REV_BLOCK := 'UT00801';
   AI_RAW_8309.revInfo.REV_NUMBER := '001.000';
   AI_RAW_8309.revInfo.REV_DATE := '2024-04-09';
   AI_RAW_8309.revInfo.REV_AUTHOR := 'M. Gledhill';
   AI_RAW_8309.___________0010_0 := false;
   AI_RAW_8309.___________0010_1 := false;
   AI_RAW_8309.AI_CODE := 16#8309;
   AI_RAW_8309.___________0020_0 := false;
   AI_RAW_8309.___________0020_1 := false;
   AI_RAW_8309.RAW_MIN := -12000;
   AI_RAW_8309.RAW_MAX := 13000;
   AI_RAW_8309.RAW_DESC := 'Thermal Resistance - 3-wire (Pt1000 climate - 392)';
   AI_RAW_8309.___________0030_1 := false;
   AI_RAW_8309.___________0030_2 := false;
   AI_RAW_8309.PARAM_TYPE := 16#08;
   AI_RAW_8309.PARAM_RANGE := 16#09;
   AI_RAW_8309.PARAM_COEF := 16#03;
   AI_RAW_8309.___________0040_1 := false;
   AI_RAW_8309.___________0040_2 := false;
   AI_RAW_8309.VALUE_COEF := 0.00392;
   AI_RAW_8005.revInfo.REV_BLOCK := 'UT00801';
   AI_RAW_8005.revInfo.REV_NUMBER := '001.000';
   AI_RAW_8005.revInfo.REV_DATE := '2024-04-09';
   AI_RAW_8005.revInfo.REV_AUTHOR := 'M. Gledhill';
   AI_RAW_8005.___________0010_0 := false;
   AI_RAW_8005.___________0010_1 := false;
   AI_RAW_8005.AI_CODE := 16#8005;
   AI_RAW_8005.___________0020_0 := false;
   AI_RAW_8005.___________0020_1 := false;
   AI_RAW_8005.RAW_MIN := -2000;
   AI_RAW_8005.RAW_MAX := 8500;
   AI_RAW_8005.RAW_DESC := 'Thermal Resistance - 3-wire (Pt1000 standard - 3851)';
   AI_RAW_8005.___________0030_1 := false;
   AI_RAW_8005.___________0030_2 := false;
   AI_RAW_8005.PARAM_TYPE := 16#08;
   AI_RAW_8005.PARAM_RANGE := 16#05;
   AI_RAW_8005.PARAM_COEF := 16#00;
   AI_RAW_8005.___________0040_1 := false;
   AI_RAW_8005.___________0040_2 := false;
   AI_RAW_8005.VALUE_COEF := 0.003851;
   AI_RAW_8205.revInfo.REV_BLOCK := 'UT00801';
   AI_RAW_8205.revInfo.REV_NUMBER := '001.000';
   AI_RAW_8205.revInfo.REV_DATE := '2024-04-09';
   AI_RAW_8205.revInfo.REV_AUTHOR := 'M. Gledhill';
   AI_RAW_8205.___________0010_0 := false;
   AI_RAW_8205.___________0010_1 := false;
   AI_RAW_8205.AI_CODE := 16#8205;
   AI_RAW_8205.___________0020_0 := false;
   AI_RAW_8205.___________0020_1 := false;
   AI_RAW_8205.RAW_MIN := -2000;
   AI_RAW_8205.RAW_MAX := 8500;
   AI_RAW_8205.RAW_DESC := 'Thermal Resistance - 3-wire (Pt1000 standard - 3902)';
   AI_RAW_8205.___________0030_1 := false;
   AI_RAW_8205.___________0030_2 := false;
   AI_RAW_8205.PARAM_TYPE := 16#08;
   AI_RAW_8205.PARAM_RANGE := 16#05;
   AI_RAW_8205.PARAM_COEF := 16#02;
   AI_RAW_8205.___________0040_1 := false;
   AI_RAW_8205.___________0040_2 := false;
   AI_RAW_8205.VALUE_COEF := 0.003902;
   AI_RAW_8505.revInfo.REV_BLOCK := 'UT00801';
   AI_RAW_8505.revInfo.REV_NUMBER := '001.000';
   AI_RAW_8505.revInfo.REV_DATE := '2024-04-09';
   AI_RAW_8505.revInfo.REV_AUTHOR := 'M. Gledhill';
   AI_RAW_8505.___________0010_0 := false;
   AI_RAW_8505.___________0010_1 := false;
   AI_RAW_8505.AI_CODE := 16#8505;
   AI_RAW_8505.___________0020_0 := false;
   AI_RAW_8505.___________0020_1 := false;
   AI_RAW_8505.RAW_MIN := -2000;
   AI_RAW_8505.RAW_MAX := 8500;
   AI_RAW_8505.RAW_DESC := 'Thermal Resistance - 3-wire (Pt1000 standard - 391)';
   AI_RAW_8505.___________0030_1 := false;
   AI_RAW_8505.___________0030_2 := false;
   AI_RAW_8505.PARAM_TYPE := 16#08;
   AI_RAW_8505.PARAM_RANGE := 16#05;
   AI_RAW_8505.PARAM_COEF := 16#05;
   AI_RAW_8505.___________0040_1 := false;
   AI_RAW_8505.___________0040_2 := false;
   AI_RAW_8505.VALUE_COEF := 0.00391;
   AI_RAW_8105.revInfo.REV_BLOCK := 'UT00801';
   AI_RAW_8105.revInfo.REV_NUMBER := '001.000';
   AI_RAW_8105.revInfo.REV_DATE := '2024-04-09';
   AI_RAW_8105.revInfo.REV_AUTHOR := 'M. Gledhill';
   AI_RAW_8105.___________0010_0 := false;
   AI_RAW_8105.___________0010_1 := false;
   AI_RAW_8105.AI_CODE := 16#8105;
   AI_RAW_8105.___________0020_0 := false;
   AI_RAW_8105.___________0020_1 := false;
   AI_RAW_8105.RAW_MIN := -2000;
   AI_RAW_8105.RAW_MAX := 8500;
   AI_RAW_8105.RAW_DESC := 'Thermal Resistance - 3-wire (Pt1000 standard - 3916)';
   AI_RAW_8105.___________0030_1 := false;
   AI_RAW_8105.___________0030_2 := false;
   AI_RAW_8105.PARAM_TYPE := 16#08;
   AI_RAW_8105.PARAM_RANGE := 16#05;
   AI_RAW_8105.PARAM_COEF := 16#01;
   AI_RAW_8105.___________0040_1 := false;
   AI_RAW_8105.___________0040_2 := false;
   AI_RAW_8105.VALUE_COEF := 0.003916;
   AI_RAW_8305.revInfo.REV_BLOCK := 'UT00801';
   AI_RAW_8305.revInfo.REV_NUMBER := '001.000';
   AI_RAW_8305.revInfo.REV_DATE := '2024-04-09';
   AI_RAW_8305.revInfo.REV_AUTHOR := 'M. Gledhill';
   AI_RAW_8305.___________0010_0 := false;
   AI_RAW_8305.___________0010_1 := false;
   AI_RAW_8305.AI_CODE := 16#8305;
   AI_RAW_8305.___________0020_0 := false;
   AI_RAW_8305.___________0020_1 := false;
   AI_RAW_8305.RAW_MIN := -2000;
   AI_RAW_8305.RAW_MAX := 8500;
   AI_RAW_8305.RAW_DESC := 'Thermal Resistance - 3-wire (Pt1000 standard - 392)';
   AI_RAW_8305.___________0030_1 := false;
   AI_RAW_8305.___________0030_2 := false;
   AI_RAW_8305.PARAM_TYPE := 16#08;
   AI_RAW_8305.PARAM_RANGE := 16#05;
   AI_RAW_8305.PARAM_COEF := 16#03;
   AI_RAW_8305.___________0040_1 := false;
   AI_RAW_8305.___________0040_2 := false;
   AI_RAW_8305.VALUE_COEF := 0.00392;
   AI_RAW_A000.revInfo.REV_BLOCK := 'UT00801';
   AI_RAW_A000.revInfo.REV_NUMBER := '001.000';
   AI_RAW_A000.revInfo.REV_DATE := '2024-04-09';
   AI_RAW_A000.revInfo.REV_AUTHOR := 'M. Gledhill';
   AI_RAW_A000.___________0010_0 := false;
   AI_RAW_A000.___________0010_1 := false;
   AI_RAW_A000.AI_CODE := 16#A000;
   AI_RAW_A000.___________0020_0 := false;
   AI_RAW_A000.___________0020_1 := false;
   AI_RAW_A000.RAW_MIN := 2500;
   AI_RAW_A000.RAW_MAX := 18200;
   AI_RAW_A000.RAW_DESC := 'Thermocouple (Type B)';
   AI_RAW_A000.___________0030_1 := false;
   AI_RAW_A000.___________0030_2 := false;
   AI_RAW_A000.PARAM_TYPE := 16#0A;
   AI_RAW_A000.PARAM_RANGE := 16#00;
   AI_RAW_A000.PARAM_COEF := 16#00;
   AI_RAW_A000.___________0040_1 := false;
   AI_RAW_A000.___________0040_2 := false;
   AI_RAW_A000.VALUE_COEF := 0.0;
   AI_RAW_A00A.revInfo.REV_BLOCK := 'UT00801';
   AI_RAW_A00A.revInfo.REV_NUMBER := '001.000';
   AI_RAW_A00A.revInfo.REV_DATE := '2024-04-09';
   AI_RAW_A00A.revInfo.REV_AUTHOR := 'M. Gledhill';
   AI_RAW_A00A.___________0010_0 := false;
   AI_RAW_A00A.___________0010_1 := false;
   AI_RAW_A00A.AI_CODE := 16#A00A;
   AI_RAW_A00A.___________0020_0 := false;
   AI_RAW_A00A.___________0020_1 := false;
   AI_RAW_A00A.RAW_MIN := 0;
   AI_RAW_A00A.RAW_MAX := 23000;
   AI_RAW_A00A.RAW_DESC := 'Thermocouple (Type C)';
   AI_RAW_A00A.___________0030_1 := false;
   AI_RAW_A00A.___________0030_2 := false;
   AI_RAW_A00A.PARAM_TYPE := 16#0A;
   AI_RAW_A00A.PARAM_RANGE := 16#0A;
   AI_RAW_A00A.PARAM_COEF := 16#00;
   AI_RAW_A00A.___________0040_1 := false;
   AI_RAW_A00A.___________0040_2 := false;
   AI_RAW_A00A.VALUE_COEF := 0.0;
   AI_RAW_A002.revInfo.REV_BLOCK := 'UT00801';
   AI_RAW_A002.revInfo.REV_NUMBER := '001.000';
   AI_RAW_A002.revInfo.REV_DATE := '2024-04-09';
   AI_RAW_A002.revInfo.REV_AUTHOR := 'M. Gledhill';
   AI_RAW_A002.___________0010_0 := false;
   AI_RAW_A002.___________0010_1 := false;
   AI_RAW_A002.AI_CODE := 16#A002;
   AI_RAW_A002.___________0020_0 := false;
   AI_RAW_A002.___________0020_1 := false;
   AI_RAW_A002.RAW_MIN := -2700;
   AI_RAW_A002.RAW_MAX := 10000;
   AI_RAW_A002.RAW_DESC := 'Thermocouple (Type E)';
   AI_RAW_A002.___________0030_1 := false;
   AI_RAW_A002.___________0030_2 := false;
   AI_RAW_A002.PARAM_TYPE := 16#0A;
   AI_RAW_A002.PARAM_RANGE := 16#02;
   AI_RAW_A002.PARAM_COEF := 16#00;
   AI_RAW_A002.___________0040_1 := false;
   AI_RAW_A002.___________0040_2 := false;
   AI_RAW_A002.VALUE_COEF := 0.0;
   AI_RAW_A005.revInfo.REV_BLOCK := 'UT00801';
   AI_RAW_A005.revInfo.REV_NUMBER := '001.000';
   AI_RAW_A005.revInfo.REV_DATE := '2024-04-09';
   AI_RAW_A005.revInfo.REV_AUTHOR := 'M. Gledhill';
   AI_RAW_A005.___________0010_0 := false;
   AI_RAW_A005.___________0010_1 := false;
   AI_RAW_A005.AI_CODE := 16#A005;
   AI_RAW_A005.___________0020_0 := false;
   AI_RAW_A005.___________0020_1 := false;
   AI_RAW_A005.RAW_MIN := -2100;
   AI_RAW_A005.RAW_MAX := 12000;
   AI_RAW_A005.RAW_DESC := 'Thermocouple (Type J)';
   AI_RAW_A005.___________0030_1 := false;
   AI_RAW_A005.___________0030_2 := false;
   AI_RAW_A005.PARAM_TYPE := 16#0A;
   AI_RAW_A005.PARAM_RANGE := 16#05;
   AI_RAW_A005.PARAM_COEF := 16#00;
   AI_RAW_A005.___________0040_1 := false;
   AI_RAW_A005.___________0040_2 := false;
   AI_RAW_A005.VALUE_COEF := 0.0;
   AI_RAW_A008.revInfo.REV_BLOCK := 'UT00801';
   AI_RAW_A008.revInfo.REV_NUMBER := '001.000';
   AI_RAW_A008.revInfo.REV_DATE := '2024-04-09';
   AI_RAW_A008.revInfo.REV_AUTHOR := 'M. Gledhill';
   AI_RAW_A008.___________0010_0 := false;
   AI_RAW_A008.___________0010_1 := false;
   AI_RAW_A008.AI_CODE := 16#A008;
   AI_RAW_A008.___________0020_0 := false;
   AI_RAW_A008.___________0020_1 := false;
   AI_RAW_A008.RAW_MIN := -2700;
   AI_RAW_A008.RAW_MAX := 13720;
   AI_RAW_A008.RAW_DESC := 'Thermocouple (Type K)';
   AI_RAW_A008.___________0030_1 := false;
   AI_RAW_A008.___________0030_2 := false;
   AI_RAW_A008.PARAM_TYPE := 16#0A;
   AI_RAW_A008.PARAM_RANGE := 16#08;
   AI_RAW_A008.PARAM_COEF := 16#00;
   AI_RAW_A008.___________0040_1 := false;
   AI_RAW_A008.___________0040_2 := false;
   AI_RAW_A008.VALUE_COEF := 0.0;
   AI_RAW_A001.revInfo.REV_BLOCK := 'UT00801';
   AI_RAW_A001.revInfo.REV_NUMBER := '001.000';
   AI_RAW_A001.revInfo.REV_DATE := '2024-04-09';
   AI_RAW_A001.revInfo.REV_AUTHOR := 'M. Gledhill';
   AI_RAW_A001.___________0010_0 := false;
   AI_RAW_A001.___________0010_1 := false;
   AI_RAW_A001.AI_CODE := 16#A001;
   AI_RAW_A001.___________0020_0 := false;
   AI_RAW_A001.___________0020_1 := false;
   AI_RAW_A001.RAW_MIN := -2700;
   AI_RAW_A001.RAW_MAX := 13000;
   AI_RAW_A001.RAW_DESC := 'Thermocouple (Type N)';
   AI_RAW_A001.___________0030_1 := false;
   AI_RAW_A001.___________0030_2 := false;
   AI_RAW_A001.PARAM_TYPE := 16#0A;
   AI_RAW_A001.PARAM_RANGE := 16#01;
   AI_RAW_A001.PARAM_COEF := 16#00;
   AI_RAW_A001.___________0040_1 := false;
   AI_RAW_A001.___________0040_2 := false;
   AI_RAW_A001.VALUE_COEF := 0.0;
   AI_RAW_A003.revInfo.REV_BLOCK := 'UT00801';
   AI_RAW_A003.revInfo.REV_NUMBER := '001.000';
   AI_RAW_A003.revInfo.REV_DATE := '2024-04-09';
   AI_RAW_A003.revInfo.REV_AUTHOR := 'M. Gledhill';
   AI_RAW_A003.___________0010_0 := false;
   AI_RAW_A003.___________0010_1 := false;
   AI_RAW_A003.AI_CODE := 16#A003;
   AI_RAW_A003.___________0020_0 := false;
   AI_RAW_A003.___________0020_1 := false;
   AI_RAW_A003.RAW_MIN := -500;
   AI_RAW_A003.RAW_MAX := 17690;
   AI_RAW_A003.RAW_DESC := 'Thermocouple (Type R)';
   AI_RAW_A003.___________0030_1 := false;
   AI_RAW_A003.___________0030_2 := false;
   AI_RAW_A003.PARAM_TYPE := 16#0A;
   AI_RAW_A003.PARAM_RANGE := 16#03;
   AI_RAW_A003.PARAM_COEF := 16#00;
   AI_RAW_A003.___________0040_1 := false;
   AI_RAW_A003.___________0040_2 := false;
   AI_RAW_A003.VALUE_COEF := 0.0;
   AI_RAW_A004.revInfo.REV_BLOCK := 'UT00801';
   AI_RAW_A004.revInfo.REV_NUMBER := '001.000';
   AI_RAW_A004.revInfo.REV_DATE := '2024-04-09';
   AI_RAW_A004.revInfo.REV_AUTHOR := 'M. Gledhill';
   AI_RAW_A004.___________0010_0 := false;
   AI_RAW_A004.___________0010_1 := false;
   AI_RAW_A004.AI_CODE := 16#A004;
   AI_RAW_A004.___________0020_0 := false;
   AI_RAW_A004.___________0020_1 := false;
   AI_RAW_A004.RAW_MIN := -500;
   AI_RAW_A004.RAW_MAX := 17690;
   AI_RAW_A004.RAW_DESC := 'Thermocouple (Type S)';
   AI_RAW_A004.___________0030_1 := false;
   AI_RAW_A004.___________0030_2 := false;
   AI_RAW_A004.PARAM_TYPE := 16#0A;
   AI_RAW_A004.PARAM_RANGE := 16#04;
   AI_RAW_A004.PARAM_COEF := 16#00;
   AI_RAW_A004.___________0040_1 := false;
   AI_RAW_A004.___________0040_2 := false;
   AI_RAW_A004.VALUE_COEF := 0.0;
   AI_RAW_A007.revInfo.REV_BLOCK := 'UT00801';
   AI_RAW_A007.revInfo.REV_NUMBER := '001.000';
   AI_RAW_A007.revInfo.REV_DATE := '2024-04-09';
   AI_RAW_A007.revInfo.REV_AUTHOR := 'M. Gledhill';
   AI_RAW_A007.___________0010_0 := false;
   AI_RAW_A007.___________0010_1 := false;
   AI_RAW_A007.AI_CODE := 16#A007;
   AI_RAW_A007.___________0020_0 := false;
   AI_RAW_A007.___________0020_1 := false;
   AI_RAW_A007.RAW_MIN := -2700;
   AI_RAW_A007.RAW_MAX := 4000;
   AI_RAW_A007.RAW_DESC := 'Thermocouple (Type T)';
   AI_RAW_A007.___________0030_1 := false;
   AI_RAW_A007.___________0030_2 := false;
   AI_RAW_A007.PARAM_TYPE := 16#0A;
   AI_RAW_A007.PARAM_RANGE := 16#07;
   AI_RAW_A007.PARAM_COEF := 16#00;
   AI_RAW_A007.___________0040_1 := false;
   AI_RAW_A007.___________0040_2 := false;
   AI_RAW_A007.VALUE_COEF := 0.0;
   AI_RAW_A00B.revInfo.REV_BLOCK := 'UT00801';
   AI_RAW_A00B.revInfo.REV_NUMBER := '001.000';
   AI_RAW_A00B.revInfo.REV_DATE := '2024-04-09';
   AI_RAW_A00B.revInfo.REV_AUTHOR := 'M. Gledhill';
   AI_RAW_A00B.___________0010_0 := false;
   AI_RAW_A00B.___________0010_1 := false;
   AI_RAW_A00B.AI_CODE := 16#A00B;
   AI_RAW_A00B.___________0020_0 := false;
   AI_RAW_A00B.___________0020_1 := false;
   AI_RAW_A00B.RAW_MIN := -2000;
   AI_RAW_A00B.RAW_MAX := 8000;
   AI_RAW_A00B.RAW_DESC := 'Thermocouple (Type TXK/XCL)';
   AI_RAW_A00B.___________0030_1 := false;
   AI_RAW_A00B.___________0030_2 := false;
   AI_RAW_A00B.PARAM_TYPE := 16#0A;
   AI_RAW_A00B.PARAM_RANGE := 16#0B;
   AI_RAW_A00B.PARAM_COEF := 16#00;
   AI_RAW_A00B.___________0040_1 := false;
   AI_RAW_A00B.___________0040_2 := false;
   AI_RAW_A00B.VALUE_COEF := 0.0;
END_DATA_BLOCK

DATA_BLOCK "DB00802_St_ConstAqRawData"   // DB802
TITLE = Static DB [SYSTEM CONSTANTS] — Analog Input Card Types, Ranges and Parameters
{ S7_Optimized_Access := 'TRUE' }
AUTHOR : M_Gledhill
FAMILY : SysConstants
NAME : St_ConstAqRawData
VERSION : 1.0
// PRACTICAL SERIES AUTOMATION LIBRARY (PAL)   —   COPYRIGHT 2020 – M. GLEDHILL (MIT LICENCE)
//                   ———— ◆ ————
// FULL ONLINE DOCUMENTATION IS AVAILABLE AT: https://practicalseries.com/2001-pal/index.html
// stored: AutoNumber false, DBAccessibleFromOPCUA true, IsOnlyStoredInLoadMemory false, IsRetainMemResEnabled false, IsWriteProtectedInAS false, MemoryReserve 100
   VAR
      _DB_Header { ExternalAccessible := 'False'; ExternalVisible := 'False'; ExternalWritable := 'False'} : Array[0..79] of Bool;   // Static DB [SYSTEM CONSTANTS] — Analog Output Card Type, Range and Parameters
      __________0000_0 { ExternalAccessible := 'False'; ExternalVisible := 'False'; ExternalWritable := 'False'} : Bool := false;
      __________0000_1 { ExternalAccessible := 'False'; ExternalVisible := 'False'; ExternalWritable := 'False'} : Bool := false;
      revInfo { ExternalWritable := 'False'} : "UT01000_St_SysRevision";
      __________0010_0 { ExternalAccessible := 'False'; ExternalVisible := 'False'; ExternalWritable := 'False'} : Bool := false;
      __________0010_1 { ExternalAccessible := 'False'; ExternalVisible := 'False'; ExternalWritable := 'False'} : Bool := false;
      AQ_RAW_0000 { ExternalWritable := 'False'} : "UT00802_St_ConstAqRawData";   // AQ User defined signal type
      __________0020_0 { ExternalAccessible := 'False'; ExternalVisible := 'False'; ExternalWritable := 'False'} : Bool := false;
      __________0020_1 { ExternalAccessible := 'False'; ExternalVisible := 'False'; ExternalWritable := 'False'} : Bool := false;   // ▀▀▀▀ ANALOG INPUT SIGNAL — VOLTAGE
      AQ_RAW_1000 { ExternalWritable := 'False'} : "UT00802_St_ConstAqRawData";   // AQ Voltage (-10 V to +10 V)
      AQ_RAW_1001 { ExternalWritable := 'False'} : "UT00802_St_ConstAqRawData";   // AQ Voltage (-5 V to +5 V)
      AQ_RAW_1002 { ExternalWritable := 'False'} : "UT00802_St_ConstAqRawData";   // AQ Voltage (0 V to 10 V)
      AQ_RAW_1003 { ExternalWritable := 'False'} : "UT00802_St_ConstAqRawData";   // AQ Voltage (1 V to 5 V)
      __________0030_0 { ExternalAccessible := 'False'; ExternalVisible := 'False'; ExternalWritable := 'False'} : Bool;
      __________0030_1 { ExternalAccessible := 'False'; ExternalVisible := 'False'; ExternalWritable := 'False'} : Bool;   // ▀▀▀▀ ANALOG INPUT SIGNAL — CURRENT
      AQ_RAW_2000 { ExternalWritable := 'False'; S7_SetPoint := 'True'} : "UT00802_St_ConstAqRawData";   // AQ Current (-20 mA to +20 mA)
      AQ_RAW_2001 { ExternalWritable := 'False'; S7_SetPoint := 'True'} : "UT00802_St_ConstAqRawData";   // AQ Current (0 mA to 20 mA)
      AQ_RAW_2002 { ExternalWritable := 'False'; S7_SetPoint := 'True'} : "UT00802_St_ConstAqRawData";   // AQ Current (4 mA to 20 mA)
   END_VAR
BEGIN
   // _DB_Header[0] : ▄▄▄▄▄▄▄▄▄▄▄▄▄▄▄▄▄▄▄▄▄▄▄▄▄▄▄▄▄▄▄▄ ＣＯＮＳＴＡＮＴＳ ▄▄
   // _DB_Header[2] : TITLE: SYSTEM CONSTANTS — ANALOG OUTPUT CARD TYPE, RANGE AND PARAMETERS
   // _DB_Header[4] : ▀▀▀▀▀▀▀▀▀▀▀▀▀▀▀▀▀▀▀▀▀▀▀▀▀▀▀▀▀▀▀▀▀▀▀▀▀▀▀▀▀▀▀▀
   // _DB_Header[5] : TYPE: STATIC
   // _DB_Header[6] : ▄▄▄▄▄▄▄▄▄▄▄▄▄▄▄▄▄▄▄▄▄▄▄▄▄▄▄▄▄▄▄▄▄▄▄▄▄▄▄▄ ʷᴵᴰ⁻ᵈʰᵐ ▄
   // _DB_Header[8] : DB00802_St_ConstAqRawData is a static data block that holds a full set of range, parameter and
   // _DB_Header[9] : descriptive data for all types of analog output card channels.
   // _DB_Header[11] : Each dataset is stored in a structure of user data type: UT00802_St_ConstAqRawData. This structure
   // _DB_Header[12] : is configured to hold all the data required by the card itself, any module accessing an analog output
   // _DB_Header[13] : and any supervisory system that is to display the type and configuration of the output channel.
   // _DB_Header[15] : All the channel data is stored as constants and is used by all modules that have an interface
   // _DB_Header[16] : to an analog output card.
   // _DB_Header[18] : The purpose of the user data type and associated data block is to provide a consistent and
   // _DB_Header[19] : tested set of range, parameter and descriptive data that can be used directly by modules that
   // _DB_Header[20] : interface with analog output cards.
   // _DB_Header[22] : The ranges correspond to the numerical values required by the card for a given type of analog card
   // _DB_Header[23] : signal. For example, a 4-20 mA card requires a numerical value of 0 to generate an output of
   // _DB_Header[24] : 4 mA ranging up to a value of 27648 at 20 mA. The data specified in the UT00802 variable would
   // _DB_Header[25] : have a lower limit of 0 and an upper limit of 27648.
   // _DB_Header[27] : In addition, each dataset contains the parametric data that defines the particular channel type and
   // _DB_Header[28] : can be used to set a particular analog output channel to a particular type and range during
   // _DB_Header[29] : runtime. Each dataset also contains a textual description of the channel type,
   // _DB_Header[30] : e.g. Current (4 mA to 20 mA)
   // _DB_Header[31] : for display and information purposes.
   // _DB_Header[33] : The PDF version of the SMDS for this module is avAQlable online here:
   // _DB_Header[34] : http://psop.uk/pal-smds-db00802-p
   // _DB_Header[36] : ━━━ ⬙⬙⬙⬙⬙⬙ ━━━
   // _DB_Header[38] : ▄▄▄▄▄▄▄▄▄▄▄▄▄▄▄▄▄▄▄▄▄▄▄▄▄▄▄▄▄▄▄▄▄▄▄▄▄▄▄▄▄▄▄▄
   // _DB_Header[39] : MODIFICATION HISTORY
   // _DB_Header[41] : This is a summary of the recent software modifications made to this block (most recent at top)
   // _DB_Header[43] : ―――――――――――――――――――――――――――――――――――――――――――
   // _DB_Header[44] : DATE REVISION MASTER BRANCH DEV
   // _DB_Header[45] : (nnn.amm) COMMIT TAG (Base ---> Merge) BRANCH Author
   // _DB_Header[46] : ———————————————————————————————————————————
   // _DB_Header[47] : 2022.05.17 001.000 D0018 D0017 D0018 None M. Gledhill
   // _DB_Header[48] : DB00802 — RELEASED FOR USE
   // _DB_Header[49] : Merge back to master branch
   // _DB_Header[51] : 2024.05.17 001.000 D0017A-000.106 D0017 N/A D0017A M. Gledhill
   // _DB_Header[52] : DB00802 Block created
   // _DB_Header[54] : 2024.05.03 000.801 D0017A-000.102 D0017 N/A D0017A M. Gledhill
   // _DB_Header[55] : DB00802 Block populated
   // _DB_Header[57] : 2024.04.09 000.101 D0017A-000.101 D0017 N/A D0017A M. Gledhill
   // _DB_Header[58] : DB00802 Block created
   // _DB_Header[59] : ———————————————————————————————————————————
   // _DB_Header[60] : Where: nnn = Major revision
   // _DB_Header[61] : a = Type (1-7 Development, 8 Proving, 9 Qualification, 0 Release)
   // _DB_Header[62] : mm = Minor revision (must be 00 if a = 0)
   // _DB_Header[63] : Block properties version number should be set to nn.a (only one decimal place)
   // _DB_Header[65] : ██████████████ █ █ █ █ END █ █ █ █ ██████████████
   revInfo.REV_BLOCK := 'DB00802';
   revInfo.REV_NUMBER := '001.000';
   revInfo.REV_DATE := '2024-05-17';
   revInfo.REV_AUTHOR := 'M. Gledhill';
   // AQ_RAW_0000.RAW_DESC : Signal type description (plAQn English)
   AQ_RAW_1000.AQ_CODE := 16#1000;
   AQ_RAW_1000.RAW_MIN := -27648;
   AQ_RAW_1000.RAW_MAX := 27648;
   AQ_RAW_1000.RAW_DESC := 'Voltage (-10 V to +10 V)';   // Signal type description (plAQn English)
   AQ_RAW_1000.PARAM_TYPE := 16#01;
   AQ_RAW_1000.PARAM_RANGE := 16#00;
   AQ_RAW_1001.AQ_CODE := 16#1001;
   AQ_RAW_1001.RAW_MIN := -27648;
   AQ_RAW_1001.RAW_MAX := 27648;
   AQ_RAW_1001.RAW_DESC := 'Voltage (-5 V to +5 V)';   // Signal type description (plAQn English)
   AQ_RAW_1001.PARAM_TYPE := 16#01;
   AQ_RAW_1001.PARAM_RANGE := 16#01;
   AQ_RAW_1002.AQ_CODE := 16#1002;
   AQ_RAW_1002.RAW_MIN := 0;
   AQ_RAW_1002.RAW_MAX := 27648;
   AQ_RAW_1002.RAW_DESC := 'Voltage (0 V to 10 V)';   // Signal type description (plAQn English)
   AQ_RAW_1002.PARAM_TYPE := 16#01;
   AQ_RAW_1002.PARAM_RANGE := 16#02;
   AQ_RAW_1003.AQ_CODE := 16#1003;
   AQ_RAW_1003.RAW_MIN := 0;
   AQ_RAW_1003.RAW_MAX := 27648;
   AQ_RAW_1003.RAW_DESC := 'Voltage (1 V to 5 V)';   // Signal type description (plAQn English)
   AQ_RAW_1003.PARAM_TYPE := 16#01;
   AQ_RAW_1003.PARAM_RANGE := 16#03;
   AQ_RAW_2000.AQ_CODE := 16#2000;
   AQ_RAW_2000.RAW_MIN := -27648;
   AQ_RAW_2000.RAW_MAX := 27648;
   AQ_RAW_2000.RAW_DESC := 'Current (-20 mA to +20 mA)';
   AQ_RAW_2000.PARAM_TYPE := 16#02;
   AQ_RAW_2000.PARAM_RANGE := 16#00;
   AQ_RAW_2001.AQ_CODE := 16#2001;
   AQ_RAW_2001.RAW_MIN := 0;
   AQ_RAW_2001.RAW_MAX := 27648;
   AQ_RAW_2001.RAW_DESC := 'Current (0 mA to 20 mA)';
   AQ_RAW_2001.PARAM_TYPE := 16#02;
   AQ_RAW_2001.PARAM_RANGE := 16#01;
   AQ_RAW_2002.AQ_CODE := 16#2002;
   AQ_RAW_2002.___________0020_0 := false;
   AQ_RAW_2002.___________0020_1 := false;
   AQ_RAW_2002.RAW_MIN := 0;
   AQ_RAW_2002.RAW_MAX := 27648;
   AQ_RAW_2002.RAW_DESC := 'Current (4 mA to 20 mA)';
   AQ_RAW_2002.PARAM_TYPE := 16#02;
   AQ_RAW_2002.PARAM_RANGE := 16#02;
END_DATA_BLOCK

